KUKA KRL program: A_40mm_helical_45_10-LIN.src

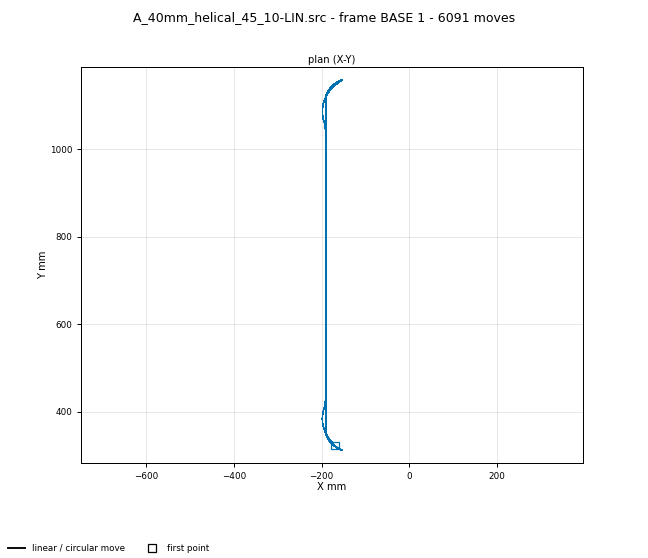
[picture p0: tool path of A_40mm_helical_45_10-LIN.src in frame BASE 1, 6091 of 6092 moves have a stored position in this frame; points joined in program order, loops and branches not executed]
&ACCESS RVP
DEF hoop( )

INTERRUPT DECL 3 WHEN $STOPMESS==TRUE DO IR_STOPM ( )
INTERRUPT ON 3
BAS (#INITMOV,0 )

ACTION(#AXIS_RESET,34,1000,#NOERROR,ERROR_CODE)
$H_POS=XHOME
PDAT_ACT=PDEFAULT
BAS (#PTP_DAT )
FDAT_ACT=FHOME
BAS (#FRAMES )
BAS (#VEL_PTP,100 )
PTP  XHOME
BAS(#TOOL,1)
BAS(#BASE,1)
LIN {X -170.340,Y +322.684,Z +0.000,A +20.000,E1 -17.457,E3 +0.000,E4 +0.000}
HALT
ACTION(#HUMM3_START,100,1000,#STOPONERROR,ERROR_CODE)
$APO.CDIS=85
$VEL_EXTAX[1]=100
LIN {X -175.568,Y +329.106,Z +0.000,A +20.000,E1 -24.747,E3 +17.234,E4 +0.000} C_DIS
LIN {X -184.074,Y +340.065,Z +0.000,A +20.000,E1 -33.664,E3 +40.174,E4 +0.000} C_DIS
LIN {X -190.779,Y +351.388,Z +0.000,A +20.000,E1 -40.083,E3 +57.952,E4 +0.000} C_DIS
LIN {X -195.254,Y +362.955,Z +0.000,A +20.000,E1 -44.515,E3 +72.705,E4 +0.000} C_DIS
LIN {X -197.754,Y +374.780,Z +0.000,A +20.000,E1 -47.450,E3 +86.127,E4 +0.000} C_DIS
LIN {X -198.310,Y +383.215,Z +0.000,A +19.956,E1 -48.698,E3 +95.251,E4 +0.000} C_DIS
LIN {X -197.912,Y +391.275,Z +0.000,A +18.601,E1 -49.158,E3 +103.969,E4 +0.000} C_DIS
LIN {X -196.679,Y +398.944,Z +0.000,A +13.989,E1 -48.784,E3 +112.523,E4 +0.000} C_DIS
LIN {X -194.742,Y +406.288,Z +0.000,A +8.476,E1 -48.001,E3 +121.206,E4 +0.000} C_DIS
LIN {X -192.748,Y +413.472,Z +0.000,A +3.905,E1 -47.267,E3 +130.216,E4 +0.000} C_DIS
LIN {X -191.781,Y +419.162,Z +0.000,A +1.739,E1 -46.975,E3 +137.484,E4 +0.000} C_DIS
LIN {X -190.795,Y +430.646,Z +0.000,A +0.152,E1 -46.707,E3 +152.145,E4 +0.000} C_DIS
LIN {X -190.395,Y +441.145,Z +0.000,A +0.001,E1 -46.583,E3 +165.538,E4 +0.000} C_DIS
LIN {X -190.239,Y +451.150,Z +0.000,A -0.000,E1 -46.528,E3 +178.306,E4 +0.000} C_DIS
LIN {X -190.161,Y +465.026,Z +0.000,A -0.000,E1 -46.506,E3 +196.021,E4 +0.000} C_DIS
LIN {X -190.142,Y +1057.148,Z +0.000,A -0.000,E1 -46.500,E3 +952.227,E4 +0.000} C_DIS
LIN {X -190.147,Y +1068.924,Z +0.000,A -0.000,E1 -46.499,E3 +967.268,E4 +0.000} C_DIS
LIN {X -190.159,Y +1079.072,Z +0.000,A -0.000,E1 -46.493,E3 +980.233,E4 +0.000} C_DIS
LIN {X -190.174,Y +1086.028,Z +0.000,A -0.000,E1 -46.483,E3 +989.127,E4 +0.000} C_DIS
LIN {X -190.200,Y +1096.186,Z +0.000,A -0.000,E1 -46.448,E3 +1002.131,E4 +0.000} C_DIS
LIN {X -190.154,Y +1108.998,Z +0.000,A -0.054,E1 -46.295,E3 +1018.626,E4 +0.000} C_DIS
LIN {X -189.772,Y +1119.341,Z +0.000,A -0.752,E1 -45.902,E3 +1032.164,E4 +0.000} C_DIS
LIN {X -189.097,Y +1124.276,Z +0.000,A -2.508,E1 -45.397,E3 +1038.896,E4 +0.000} C_DIS
LIN {X -187.410,Y +1129.069,Z +0.000,A -5.304,E1 -44.585,E3 +1046.069,E4 +0.000} C_DIS
LIN {X -183.899,Y +1134.873,Z +0.000,A -10.372,E1 -42.805,E3 +1056.075,E4 +0.000} C_DIS
LIN {X -179.711,Y +1140.065,Z +0.000,A -15.940,E1 -40.393,E3 +1066.861,E4 +0.000} C_DIS
LIN {X -176.763,Y +1143.197,Z +0.000,A -18.748,E1 -38.674,E3 +1074.599,E4 +0.000} C_DIS
LIN {X -172.185,Y +1147.423,Z +0.000,A -19.971,E1 -36.175,E3 +1087.329,E4 +0.000} C_DIS
LIN {X -165.999,Y +1152.127,Z +0.000,A -20.000,E1 -32.027,E3 +1107.087,E4 +0.000} C_DIS
LIN {X -160.138,Y +1155.667,Z +0.000,A -20.000,E1 -26.368,E3 +1131.457,E4 +0.000} C_DIS
LIN {X -155.625,Y +1157.756,Z +0.000,A -20.000,E1 -19.505,E3 +1160.133,E4 +0.000} C_DIS
LIN {X -153.552,Y +1158.113,Z +0.000,A -20.000,E1 -11.113,E3 +1195.884,E4 +0.000} C_DIS
LIN {X -156.311,Y +1155.540,Z +0.000,A -20.000,E1 -0.839,E3 +1239.244,E4 +0.000} C_DIS
LIN {X -161.281,Y +1151.851,Z +0.000,A -20.000,E1 +7.737,E3 +1269.143,E4 +0.000} C_DIS
LIN {X -167.493,Y +1147.157,Z +0.000,A -20.000,E1 +16.195,E3 +1293.582,E4 +0.000} C_DIS
LIN {X -173.235,Y +1142.221,Z +0.000,A -20.000,E1 +22.930,E3 +1310.884,E4 +0.000} C_DIS
LIN {X -181.123,Y +1133.734,Z +0.000,A -20.000,E1 +30.868,E3 +1331.640,E4 +0.000} C_DIS
LIN {X -189.654,Y +1120.856,Z +0.000,A -20.000,E1 +39.018,E3 +1353.654,E4 +0.000} C_DIS
LIN {X -195.246,Y +1107.046,Z +0.000,A -20.000,E1 +44.515,E3 +1371.556,E4 +0.000} C_DIS
LIN {X -198.051,Y +1092.368,Z +0.000,A -20.000,E1 +47.947,E3 +1388.082,E4 +0.000} C_DIS
LIN {X -198.143,Y +1081.370,Z +0.000,A -19.806,E1 +49.153,E3 +1399.943,E4 +0.000} C_DIS
LIN {X -197.177,Y +1073.569,Z +0.000,A -17.356,E1 +49.162,E3 +1408.527,E4 +0.000} C_DIS
LIN {X -195.448,Y +1066.139,Z +0.000,A -12.154,E1 +48.512,E3 +1417.122,E4 +0.000} C_DIS
LIN {X -193.346,Y +1058.941,Z +0.000,A -7.133,E1 +47.724,E3 +1426.002,E4 +0.000} C_DIS
LIN {X -191.781,Y +1050.839,Z +0.000,A -3.715,E1 +47.274,E3 +1436.335,E4 +0.000} C_DIS
LIN {X -190.795,Y +1039.355,Z +0.000,A -0.983,E1 +46.842,E3 +1450.995,E4 +0.000} C_DIS
LIN {X -190.395,Y +1028.856,Z +0.000,A -0.089,E1 +46.598,E3 +1464.389,E4 +0.000} C_DIS
LIN {X -190.239,Y +1018.851,Z +0.000,A -0.004,E1 +46.529,E3 +1477.157,E4 +0.000} C_DIS
LIN {X -190.161,Y +1004.975,Z +0.000,A +0.000,E1 +46.506,E3 +1494.871,E4 +0.000} C_DIS
LIN {X -190.142,Y +412.853,Z +0.000,A +0.000,E1 +46.501,E3 +2251.077,E4 +0.000} C_DIS
LIN {X -190.147,Y +401.077,Z +0.000,A +0.000,E1 +46.499,E3 +2266.118,E4 +0.000} C_DIS
LIN {X -190.159,Y +390.929,Z +0.000,A +0.000,E1 +46.494,E3 +2279.084,E4 +0.000} C_DIS
LIN {X -190.174,Y +383.973,Z +0.000,A +0.000,E1 +46.484,E3 +2287.977,E4 +0.000} C_DIS
LIN {X -190.200,Y +373.815,Z +0.000,A +0.000,E1 +46.448,E3 +2300.982,E4 +0.000} C_DIS
LIN {X -190.154,Y +361.003,Z +0.000,A +0.000,E1 +46.303,E3 +2317.476,E4 +0.000} C_DIS
LIN {X -189.772,Y +350.660,Z +0.000,A +0.049,E1 +45.996,E3 +2331.015,E4 +0.000} C_DIS
LIN {X -189.325,Y +346.917,Z +0.000,A +0.243,E1 +45.771,E3 +2336.084,E4 +0.000} C_DIS
LIN {X -188.196,Y +342.754,Z +0.000,A +1.966,E1 +45.249,E3 +2342.092,E4 +0.000} C_DIS
LIN {X -185.199,Y +337.023,Z +0.000,A +6.630,E1 +43.793,E3 +2351.466,E4 +0.000} C_DIS
LIN {X -181.141,Y +331.596,Z +0.000,A +12.274,E1 +41.569,E3 +2362.026,E4 +0.000} C_DIS
LIN {X -176.762,Y +326.804,Z +0.000,A +17.560,E1 +38.898,E3 +2373.450,E4 +0.000} C_DIS
LIN {X -172.184,Y +322.578,Z +0.000,A +19.859,E1 +36.197,E3 +2386.180,E4 +0.000} C_DIS
LIN {X -165.998,Y +317.874,Z +0.000,A +20.000,E1 +32.027,E3 +2405.938,E4 +0.000} C_DIS
LIN {X -160.137,Y +314.334,Z +0.000,A +20.000,E1 +26.368,E3 +2430.307,E4 +0.000} C_DIS
LIN {X -155.624,Y +312.245,Z +0.000,A +20.000,E1 +19.506,E3 +2458.983,E4 +0.000} C_DIS
LIN {X -153.557,Y +311.879,Z +0.000,A +20.000,E1 +11.113,E3 +2494.738,E4 +0.000} C_DIS
LIN {X -155.320,Y +313.348,Z +0.000,A +20.000,E1 +3.401,E3 +2527.922,E4 +0.000} C_DIS
LIN {X -160.005,Y +315.804,Z +0.000,A +20.000,E1 -4.720,E3 +2558.300,E4 +0.000} C_DIS
LIN {X -164.504,Y +318.255,Z +0.000,A +20.000,E1 -10.663,E3 +2577.669,E4 +0.000} C_DIS
LIN {X -170.340,Y +322.684,Z +0.000,A +20.000,E1 -17.457,E3 +2597.701,E4 +0.000} C_DIS
LIN {X -175.568,Y +329.106,Z +0.000,A +20.000,E1 -24.747,E3 +2614.935,E4 +0.000} C_DIS
LIN {X -184.074,Y +340.065,Z +0.000,A +20.000,E1 -33.664,E3 +2637.875,E4 +0.000} C_DIS
LIN {X -190.779,Y +351.388,Z +0.000,A +20.000,E1 -40.083,E3 +2655.653,E4 +0.000} C_DIS
LIN {X -195.254,Y +362.955,Z +0.000,A +20.000,E1 -44.515,E3 +2670.406,E4 +0.000} C_DIS
LIN {X -197.754,Y +374.780,Z +0.000,A +20.000,E1 -47.450,E3 +2683.828,E4 +0.000} C_DIS
LIN {X -198.310,Y +383.215,Z +0.000,A +19.956,E1 -48.698,E3 +2692.952,E4 +0.000} C_DIS
LIN {X -197.912,Y +391.275,Z +0.000,A +18.601,E1 -49.158,E3 +2701.670,E4 +0.000} C_DIS
LIN {X -196.679,Y +398.944,Z +0.000,A +13.989,E1 -48.784,E3 +2710.224,E4 +0.000} C_DIS
LIN {X -194.742,Y +406.288,Z +0.000,A +8.476,E1 -48.001,E3 +2718.907,E4 +0.000} C_DIS
LIN {X -192.748,Y +413.472,Z +0.000,A +3.905,E1 -47.267,E3 +2727.917,E4 +0.000} C_DIS
LIN {X -191.781,Y +419.162,Z +0.000,A +1.739,E1 -46.975,E3 +2735.185,E4 +0.000} C_DIS
LIN {X -190.795,Y +430.646,Z +0.000,A +0.152,E1 -46.707,E3 +2749.846,E4 +0.000} C_DIS
LIN {X -190.395,Y +441.145,Z +0.000,A +0.001,E1 -46.583,E3 +2763.239,E4 +0.000} C_DIS
LIN {X -190.239,Y +451.150,Z +0.000,A -0.000,E1 -46.528,E3 +2776.007,E4 +0.000} C_DIS
LIN {X -190.161,Y +465.026,Z +0.000,A -0.000,E1 -46.506,E3 +2793.722,E4 +0.000} C_DIS
LIN {X -190.142,Y +1057.148,Z +0.000,A -0.000,E1 -46.500,E3 +3549.928,E4 +0.000} C_DIS
LIN {X -190.147,Y +1068.924,Z +0.000,A -0.000,E1 -46.499,E3 +3564.969,E4 +0.000} C_DIS
LIN {X -190.159,Y +1079.072,Z +0.000,A -0.000,E1 -46.493,E3 +3577.934,E4 +0.000} C_DIS
LIN {X -190.174,Y +1086.028,Z +0.000,A -0.000,E1 -46.483,E3 +3586.828,E4 +0.000} C_DIS
LIN {X -190.200,Y +1096.186,Z +0.000,A -0.000,E1 -46.448,E3 +3599.832,E4 +0.000} C_DIS
LIN {X -190.154,Y +1108.998,Z +0.000,A -0.054,E1 -46.295,E3 +3616.327,E4 +0.000} C_DIS
LIN {X -189.772,Y +1119.341,Z +0.000,A -0.752,E1 -45.902,E3 +3629.865,E4 +0.000} C_DIS
LIN {X -189.097,Y +1124.276,Z +0.000,A -2.508,E1 -45.397,E3 +3636.597,E4 +0.000} C_DIS
LIN {X -187.410,Y +1129.069,Z +0.000,A -5.304,E1 -44.585,E3 +3643.770,E4 +0.000} C_DIS
LIN {X -183.899,Y +1134.873,Z +0.000,A -10.372,E1 -42.805,E3 +3653.776,E4 +0.000} C_DIS
LIN {X -179.711,Y +1140.065,Z +0.000,A -15.940,E1 -40.393,E3 +3664.562,E4 +0.000} C_DIS
LIN {X -176.763,Y +1143.197,Z +0.000,A -18.748,E1 -38.674,E3 +3672.300,E4 +0.000} C_DIS
LIN {X -172.185,Y +1147.423,Z +0.000,A -19.971,E1 -36.175,E3 +3685.030,E4 +0.000} C_DIS
LIN {X -165.999,Y +1152.127,Z +0.000,A -20.000,E1 -32.027,E3 +3704.788,E4 +0.000} C_DIS
LIN {X -160.138,Y +1155.667,Z +0.000,A -20.000,E1 -26.368,E3 +3729.158,E4 +0.000} C_DIS
LIN {X -155.625,Y +1157.756,Z +0.000,A -20.000,E1 -19.505,E3 +3757.834,E4 +0.000} C_DIS
LIN {X -153.552,Y +1158.113,Z +0.000,A -20.000,E1 -11.113,E3 +3793.585,E4 +0.000} C_DIS
LIN {X -156.311,Y +1155.540,Z +0.000,A -20.000,E1 -0.839,E3 +3836.945,E4 +0.000} C_DIS
LIN {X -161.281,Y +1151.851,Z +0.000,A -20.000,E1 +7.737,E3 +3866.844,E4 +0.000} C_DIS
LIN {X -167.493,Y +1147.157,Z +0.000,A -20.000,E1 +16.195,E3 +3891.283,E4 +0.000} C_DIS
LIN {X -173.235,Y +1142.221,Z +0.000,A -20.000,E1 +22.930,E3 +3908.585,E4 +0.000} C_DIS
LIN {X -181.123,Y +1133.734,Z +0.000,A -20.000,E1 +30.868,E3 +3929.341,E4 +0.000} C_DIS
LIN {X -189.654,Y +1120.856,Z +0.000,A -20.000,E1 +39.018,E3 +3951.355,E4 +0.000} C_DIS
LIN {X -195.246,Y +1107.046,Z +0.000,A -20.000,E1 +44.515,E3 +3969.257,E4 +0.000} C_DIS
LIN {X -198.051,Y +1092.368,Z +0.000,A -20.000,E1 +47.947,E3 +3985.783,E4 +0.000} C_DIS
LIN {X -198.143,Y +1081.370,Z +0.000,A -19.806,E1 +49.153,E3 +3997.644,E4 +0.000} C_DIS
LIN {X -197.177,Y +1073.569,Z +0.000,A -17.356,E1 +49.162,E3 +4006.228,E4 +0.000} C_DIS
LIN {X -195.448,Y +1066.139,Z +0.000,A -12.154,E1 +48.512,E3 +4014.823,E4 +0.000} C_DIS
LIN {X -193.346,Y +1058.941,Z +0.000,A -7.133,E1 +47.724,E3 +4023.703,E4 +0.000} C_DIS
LIN {X -191.781,Y +1050.839,Z +0.000,A -3.715,E1 +47.274,E3 +4034.036,E4 +0.000} C_DIS
LIN {X -190.795,Y +1039.355,Z +0.000,A -0.983,E1 +46.842,E3 +4048.696,E4 +0.000} C_DIS
LIN {X -190.395,Y +1028.856,Z +0.000,A -0.089,E1 +46.598,E3 +4062.090,E4 +0.000} C_DIS
LIN {X -190.239,Y +1018.851,Z +0.000,A -0.004,E1 +46.529,E3 +4074.858,E4 +0.000} C_DIS
LIN {X -190.161,Y +1004.975,Z +0.000,A +0.000,E1 +46.506,E3 +4092.572,E4 +0.000} C_DIS
LIN {X -190.142,Y +412.853,Z +0.000,A +0.000,E1 +46.501,E3 +4848.778,E4 +0.000} C_DIS
LIN {X -190.147,Y +401.077,Z +0.000,A +0.000,E1 +46.499,E3 +4863.819,E4 +0.000} C_DIS
LIN {X -190.159,Y +390.929,Z +0.000,A +0.000,E1 +46.494,E3 +4876.785,E4 +0.000} C_DIS
LIN {X -190.174,Y +383.973,Z +0.000,A +0.000,E1 +46.484,E3 +4885.678,E4 +0.000} C_DIS
LIN {X -190.200,Y +373.815,Z +0.000,A +0.000,E1 +46.448,E3 +4898.683,E4 +0.000} C_DIS
LIN {X -190.154,Y +361.003,Z +0.000,A +0.000,E1 +46.303,E3 +4915.177,E4 +0.000} C_DIS
LIN {X -189.772,Y +350.660,Z +0.000,A +0.049,E1 +45.996,E3 +4928.716,E4 +0.000} C_DIS
LIN {X -189.325,Y +346.917,Z +0.000,A +0.243,E1 +45.771,E3 +4933.785,E4 +0.000} C_DIS
LIN {X -188.196,Y +342.754,Z +0.000,A +1.966,E1 +45.249,E3 +4939.793,E4 +0.000} C_DIS
LIN {X -185.199,Y +337.023,Z +0.000,A +6.630,E1 +43.793,E3 +4949.167,E4 +0.000} C_DIS
LIN {X -181.141,Y +331.596,Z +0.000,A +12.274,E1 +41.569,E3 +4959.727,E4 +0.000} C_DIS
LIN {X -176.762,Y +326.804,Z +0.000,A +17.560,E1 +38.898,E3 +4971.151,E4 +0.000} C_DIS
LIN {X -172.184,Y +322.578,Z +0.000,A +19.859,E1 +36.197,E3 +4983.881,E4 +0.000} C_DIS
LIN {X -165.998,Y +317.874,Z +0.000,A +20.000,E1 +32.027,E3 +5003.639,E4 +0.000} C_DIS
LIN {X -160.137,Y +314.334,Z +0.000,A +20.000,E1 +26.368,E3 +5028.008,E4 +0.000} C_DIS
LIN {X -155.624,Y +312.245,Z +0.000,A +20.000,E1 +19.506,E3 +5056.684,E4 +0.000} C_DIS
LIN {X -153.557,Y +311.879,Z +0.000,A +20.000,E1 +11.113,E3 +5092.439,E4 +0.000} C_DIS
LIN {X -155.320,Y +313.348,Z +0.000,A +20.000,E1 +3.401,E3 +5125.623,E4 +0.000} C_DIS
LIN {X -160.005,Y +315.804,Z +0.000,A +20.000,E1 -4.720,E3 +5156.001,E4 +0.000} C_DIS
LIN {X -164.504,Y +318.255,Z +0.000,A +20.000,E1 -10.663,E3 +5175.370,E4 +0.000} C_DIS
LIN {X -170.340,Y +322.684,Z +0.000,A +20.000,E1 -17.457,E3 +5195.402,E4 +0.000} C_DIS
LIN {X -175.568,Y +329.106,Z +0.000,A +20.000,E1 -24.747,E3 +5212.636,E4 +0.000} C_DIS
LIN {X -184.074,Y +340.065,Z +0.000,A +20.000,E1 -33.664,E3 +5235.576,E4 +0.000} C_DIS
LIN {X -190.779,Y +351.388,Z +0.000,A +20.000,E1 -40.083,E3 +5253.354,E4 +0.000} C_DIS
LIN {X -195.254,Y +362.955,Z +0.000,A +20.000,E1 -44.515,E3 +5268.107,E4 +0.000} C_DIS
LIN {X -197.754,Y +374.780,Z +0.000,A +20.000,E1 -47.450,E3 +5281.529,E4 +0.000} C_DIS
LIN {X -198.310,Y +383.215,Z +0.000,A +19.956,E1 -48.698,E3 +5290.653,E4 +0.000} C_DIS
LIN {X -197.912,Y +391.275,Z +0.000,A +18.601,E1 -49.158,E3 +5299.371,E4 +0.000} C_DIS
LIN {X -196.679,Y +398.944,Z +0.000,A +13.989,E1 -48.784,E3 +5307.925,E4 +0.000} C_DIS
LIN {X -194.742,Y +406.288,Z +0.000,A +8.476,E1 -48.001,E3 +5316.608,E4 +0.000} C_DIS
LIN {X -192.748,Y +413.472,Z +0.000,A +3.905,E1 -47.267,E3 +5325.618,E4 +0.000} C_DIS
LIN {X -191.781,Y +419.162,Z +0.000,A +1.739,E1 -46.975,E3 +5332.886,E4 +0.000} C_DIS
LIN {X -190.795,Y +430.646,Z +0.000,A +0.152,E1 -46.707,E3 +5347.547,E4 +0.000} C_DIS
LIN {X -190.395,Y +441.145,Z +0.000,A +0.001,E1 -46.583,E3 +5360.940,E4 +0.000} C_DIS
LIN {X -190.239,Y +451.150,Z +0.000,A -0.000,E1 -46.528,E3 +5373.708,E4 +0.000} C_DIS
LIN {X -190.161,Y +465.026,Z +0.000,A -0.000,E1 -46.506,E3 +5391.423,E4 +0.000} C_DIS
LIN {X -190.142,Y +1057.148,Z +0.000,A -0.000,E1 -46.500,E3 +6147.629,E4 +0.000} C_DIS
LIN {X -190.147,Y +1068.924,Z +0.000,A -0.000,E1 -46.499,E3 +6162.670,E4 +0.000} C_DIS
LIN {X -190.159,Y +1079.072,Z +0.000,A -0.000,E1 -46.493,E3 +6175.635,E4 +0.000} C_DIS
LIN {X -190.174,Y +1086.028,Z +0.000,A -0.000,E1 -46.483,E3 +6184.529,E4 +0.000} C_DIS
LIN {X -190.200,Y +1096.186,Z +0.000,A -0.000,E1 -46.448,E3 +6197.533,E4 +0.000} C_DIS
LIN {X -190.154,Y +1108.998,Z +0.000,A -0.054,E1 -46.295,E3 +6214.028,E4 +0.000} C_DIS
LIN {X -189.772,Y +1119.341,Z +0.000,A -0.752,E1 -45.902,E3 +6227.566,E4 +0.000} C_DIS
LIN {X -189.097,Y +1124.276,Z +0.000,A -2.508,E1 -45.397,E3 +6234.298,E4 +0.000} C_DIS
LIN {X -187.410,Y +1129.069,Z +0.000,A -5.304,E1 -44.585,E3 +6241.471,E4 +0.000} C_DIS
LIN {X -183.899,Y +1134.873,Z +0.000,A -10.372,E1 -42.805,E3 +6251.477,E4 +0.000} C_DIS
LIN {X -179.711,Y +1140.065,Z +0.000,A -15.940,E1 -40.393,E3 +6262.263,E4 +0.000} C_DIS
LIN {X -176.763,Y +1143.197,Z +0.000,A -18.748,E1 -38.674,E3 +6270.001,E4 +0.000} C_DIS
LIN {X -172.185,Y +1147.423,Z +0.000,A -19.971,E1 -36.175,E3 +6282.731,E4 +0.000} C_DIS
LIN {X -165.999,Y +1152.127,Z +0.000,A -20.000,E1 -32.027,E3 +6302.489,E4 +0.000} C_DIS
LIN {X -160.138,Y +1155.667,Z +0.000,A -20.000,E1 -26.368,E3 +6326.859,E4 +0.000} C_DIS
LIN {X -155.625,Y +1157.756,Z +0.000,A -20.000,E1 -19.505,E3 +6355.535,E4 +0.000} C_DIS
LIN {X -153.552,Y +1158.113,Z +0.000,A -20.000,E1 -11.113,E3 +6391.286,E4 +0.000} C_DIS
LIN {X -156.311,Y +1155.540,Z +0.000,A -20.000,E1 -0.839,E3 +6434.646,E4 +0.000} C_DIS
LIN {X -161.281,Y +1151.851,Z +0.000,A -20.000,E1 +7.737,E3 +6464.545,E4 +0.000} C_DIS
LIN {X -167.493,Y +1147.157,Z +0.000,A -20.000,E1 +16.195,E3 +6488.984,E4 +0.000} C_DIS
LIN {X -173.235,Y +1142.221,Z +0.000,A -20.000,E1 +22.930,E3 +6506.286,E4 +0.000} C_DIS
LIN {X -181.123,Y +1133.734,Z +0.000,A -20.000,E1 +30.868,E3 +6527.042,E4 +0.000} C_DIS
LIN {X -189.654,Y +1120.856,Z +0.000,A -20.000,E1 +39.018,E3 +6549.056,E4 +0.000} C_DIS
LIN {X -195.246,Y +1107.046,Z +0.000,A -20.000,E1 +44.515,E3 +6566.958,E4 +0.000} C_DIS
LIN {X -198.051,Y +1092.368,Z +0.000,A -20.000,E1 +47.947,E3 +6583.484,E4 +0.000} C_DIS
LIN {X -198.143,Y +1081.370,Z +0.000,A -19.806,E1 +49.153,E3 +6595.345,E4 +0.000} C_DIS
LIN {X -197.177,Y +1073.569,Z +0.000,A -17.356,E1 +49.162,E3 +6603.929,E4 +0.000} C_DIS
LIN {X -195.448,Y +1066.139,Z +0.000,A -12.154,E1 +48.512,E3 +6612.524,E4 +0.000} C_DIS
LIN {X -193.346,Y +1058.941,Z +0.000,A -7.133,E1 +47.724,E3 +6621.404,E4 +0.000} C_DIS
LIN {X -191.781,Y +1050.839,Z +0.000,A -3.715,E1 +47.274,E3 +6631.737,E4 +0.000} C_DIS
LIN {X -190.795,Y +1039.355,Z +0.000,A -0.983,E1 +46.842,E3 +6646.397,E4 +0.000} C_DIS
LIN {X -190.395,Y +1028.856,Z +0.000,A -0.089,E1 +46.598,E3 +6659.791,E4 +0.000} C_DIS
LIN {X -190.239,Y +1018.851,Z +0.000,A -0.004,E1 +46.529,E3 +6672.559,E4 +0.000} C_DIS
LIN {X -190.161,Y +1004.975,Z +0.000,A +0.000,E1 +46.506,E3 +6690.273,E4 +0.000} C_DIS
LIN {X -190.142,Y +412.853,Z +0.000,A +0.000,E1 +46.501,E3 +7446.479,E4 +0.000} C_DIS
LIN {X -190.147,Y +401.077,Z +0.000,A +0.000,E1 +46.499,E3 +7461.520,E4 +0.000} C_DIS
LIN {X -190.159,Y +390.929,Z +0.000,A +0.000,E1 +46.494,E3 +7474.486,E4 +0.000} C_DIS
LIN {X -190.174,Y +383.973,Z +0.000,A +0.000,E1 +46.484,E3 +7483.379,E4 +0.000} C_DIS
LIN {X -190.200,Y +373.815,Z +0.000,A +0.000,E1 +46.448,E3 +7496.384,E4 +0.000} C_DIS
LIN {X -190.154,Y +361.003,Z +0.000,A +0.000,E1 +46.303,E3 +7512.878,E4 +0.000} C_DIS
LIN {X -189.772,Y +350.660,Z +0.000,A +0.049,E1 +45.996,E3 +7526.417,E4 +0.000} C_DIS
LIN {X -189.325,Y +346.917,Z +0.000,A +0.243,E1 +45.771,E3 +7531.486,E4 +0.000} C_DIS
LIN {X -188.196,Y +342.754,Z +0.000,A +1.966,E1 +45.249,E3 +7537.494,E4 +0.000} C_DIS
LIN {X -185.199,Y +337.023,Z +0.000,A +6.630,E1 +43.793,E3 +7546.868,E4 +0.000} C_DIS
LIN {X -181.141,Y +331.596,Z +0.000,A +12.274,E1 +41.569,E3 +7557.428,E4 +0.000} C_DIS
LIN {X -176.762,Y +326.804,Z +0.000,A +17.560,E1 +38.898,E3 +7568.852,E4 +0.000} C_DIS
LIN {X -172.184,Y +322.578,Z +0.000,A +19.859,E1 +36.197,E3 +7581.582,E4 +0.000} C_DIS
LIN {X -165.998,Y +317.874,Z +0.000,A +20.000,E1 +32.027,E3 +7601.340,E4 +0.000} C_DIS
LIN {X -160.137,Y +314.334,Z +0.000,A +20.000,E1 +26.368,E3 +7625.709,E4 +0.000} C_DIS
LIN {X -155.624,Y +312.245,Z +0.000,A +20.000,E1 +19.506,E3 +7654.385,E4 +0.000} C_DIS
LIN {X -153.557,Y +311.879,Z +0.000,A +20.000,E1 +11.113,E3 +7690.140,E4 +0.000} C_DIS
LIN {X -155.320,Y +313.348,Z +0.000,A +20.000,E1 +3.401,E3 +7723.324,E4 +0.000} C_DIS
LIN {X -160.005,Y +315.804,Z +0.000,A +20.000,E1 -4.720,E3 +7753.702,E4 +0.000} C_DIS
LIN {X -164.504,Y +318.255,Z +0.000,A +20.000,E1 -10.663,E3 +7773.071,E4 +0.000} C_DIS
LIN {X -170.340,Y +322.684,Z +0.000,A +20.000,E1 -17.457,E3 +7793.103,E4 +0.000} C_DIS
LIN {X -175.568,Y +329.106,Z +0.000,A +20.000,E1 -24.747,E3 +7810.337,E4 +0.000} C_DIS
LIN {X -184.074,Y +340.065,Z +0.000,A +20.000,E1 -33.664,E3 +7833.277,E4 +0.000} C_DIS
LIN {X -190.779,Y +351.388,Z +0.000,A +20.000,E1 -40.083,E3 +7851.055,E4 +0.000} C_DIS
LIN {X -195.254,Y +362.955,Z +0.000,A +20.000,E1 -44.515,E3 +7865.808,E4 +0.000} C_DIS
LIN {X -197.754,Y +374.780,Z +0.000,A +20.000,E1 -47.450,E3 +7879.230,E4 +0.000} C_DIS
LIN {X -198.310,Y +383.215,Z +0.000,A +19.956,E1 -48.698,E3 +7888.354,E4 +0.000} C_DIS
LIN {X -197.912,Y +391.275,Z +0.000,A +18.601,E1 -49.158,E3 +7897.072,E4 +0.000} C_DIS
LIN {X -196.679,Y +398.944,Z +0.000,A +13.989,E1 -48.784,E3 +7905.626,E4 +0.000} C_DIS
LIN {X -194.742,Y +406.288,Z +0.000,A +8.476,E1 -48.001,E3 +7914.309,E4 +0.000} C_DIS
LIN {X -192.748,Y +413.472,Z +0.000,A +3.905,E1 -47.267,E3 +7923.319,E4 +0.000} C_DIS
LIN {X -191.781,Y +419.162,Z +0.000,A +1.739,E1 -46.975,E3 +7930.587,E4 +0.000} C_DIS
LIN {X -190.795,Y +430.646,Z +0.000,A +0.152,E1 -46.707,E3 +7945.248,E4 +0.000} C_DIS
LIN {X -190.395,Y +441.145,Z +0.000,A +0.001,E1 -46.583,E3 +7958.641,E4 +0.000} C_DIS
LIN {X -190.239,Y +451.150,Z +0.000,A -0.000,E1 -46.528,E3 +7971.409,E4 +0.000} C_DIS
LIN {X -190.161,Y +465.026,Z +0.000,A -0.000,E1 -46.506,E3 +7989.124,E4 +0.000} C_DIS
LIN {X -190.142,Y +1057.148,Z +0.000,A -0.000,E1 -46.500,E3 +8745.330,E4 +0.000} C_DIS
LIN {X -190.147,Y +1068.924,Z +0.000,A -0.000,E1 -46.499,E3 +8760.371,E4 +0.000} C_DIS
LIN {X -190.159,Y +1079.072,Z +0.000,A -0.000,E1 -46.493,E3 +8773.336,E4 +0.000} C_DIS
LIN {X -190.174,Y +1086.028,Z +0.000,A -0.000,E1 -46.483,E3 +8782.230,E4 +0.000} C_DIS
LIN {X -190.200,Y +1096.186,Z +0.000,A -0.000,E1 -46.448,E3 +8795.234,E4 +0.000} C_DIS
LIN {X -190.154,Y +1108.998,Z +0.000,A -0.054,E1 -46.295,E3 +8811.729,E4 +0.000} C_DIS
LIN {X -189.772,Y +1119.341,Z +0.000,A -0.752,E1 -45.902,E3 +8825.267,E4 +0.000} C_DIS
LIN {X -189.097,Y +1124.276,Z +0.000,A -2.508,E1 -45.397,E3 +8831.999,E4 +0.000} C_DIS
LIN {X -187.410,Y +1129.069,Z +0.000,A -5.304,E1 -44.585,E3 +8839.172,E4 +0.000} C_DIS
LIN {X -183.899,Y +1134.873,Z +0.000,A -10.372,E1 -42.805,E3 +8849.178,E4 +0.000} C_DIS
LIN {X -179.711,Y +1140.065,Z +0.000,A -15.940,E1 -40.393,E3 +8859.964,E4 +0.000} C_DIS
LIN {X -176.763,Y +1143.197,Z +0.000,A -18.748,E1 -38.674,E3 +8867.702,E4 +0.000} C_DIS
LIN {X -172.185,Y +1147.423,Z +0.000,A -19.971,E1 -36.175,E3 +8880.432,E4 +0.000} C_DIS
LIN {X -165.999,Y +1152.127,Z +0.000,A -20.000,E1 -32.027,E3 +8900.190,E4 +0.000} C_DIS
LIN {X -160.138,Y +1155.667,Z +0.000,A -20.000,E1 -26.368,E3 +8924.560,E4 +0.000} C_DIS
LIN {X -155.625,Y +1157.756,Z +0.000,A -20.000,E1 -19.505,E3 +8953.236,E4 +0.000} C_DIS
LIN {X -153.552,Y +1158.113,Z +0.000,A -20.000,E1 -11.113,E3 +8988.987,E4 +0.000} C_DIS
LIN {X -156.311,Y +1155.540,Z +0.000,A -20.000,E1 -0.839,E3 +9032.347,E4 +0.000} C_DIS
LIN {X -161.281,Y +1151.851,Z +0.000,A -20.000,E1 +7.737,E3 +9062.246,E4 +0.000} C_DIS
LIN {X -167.493,Y +1147.157,Z +0.000,A -20.000,E1 +16.195,E3 +9086.685,E4 +0.000} C_DIS
LIN {X -173.235,Y +1142.221,Z +0.000,A -20.000,E1 +22.930,E3 +9103.987,E4 +0.000} C_DIS
LIN {X -181.123,Y +1133.734,Z +0.000,A -20.000,E1 +30.868,E3 +9124.743,E4 +0.000} C_DIS
LIN {X -189.654,Y +1120.856,Z +0.000,A -20.000,E1 +39.018,E3 +9146.757,E4 +0.000} C_DIS
LIN {X -195.246,Y +1107.046,Z +0.000,A -20.000,E1 +44.515,E3 +9164.659,E4 +0.000} C_DIS
LIN {X -198.051,Y +1092.368,Z +0.000,A -20.000,E1 +47.947,E3 +9181.185,E4 +0.000} C_DIS
LIN {X -198.143,Y +1081.370,Z +0.000,A -19.806,E1 +49.153,E3 +9193.046,E4 +0.000} C_DIS
LIN {X -197.177,Y +1073.569,Z +0.000,A -17.356,E1 +49.162,E3 +9201.630,E4 +0.000} C_DIS
LIN {X -195.448,Y +1066.139,Z +0.000,A -12.154,E1 +48.512,E3 +9210.225,E4 +0.000} C_DIS
LIN {X -193.346,Y +1058.941,Z +0.000,A -7.133,E1 +47.724,E3 +9219.105,E4 +0.000} C_DIS
LIN {X -191.781,Y +1050.839,Z +0.000,A -3.715,E1 +47.274,E3 +9229.438,E4 +0.000} C_DIS
LIN {X -190.795,Y +1039.355,Z +0.000,A -0.983,E1 +46.842,E3 +9244.098,E4 +0.000} C_DIS
LIN {X -190.395,Y +1028.856,Z +0.000,A -0.089,E1 +46.598,E3 +9257.492,E4 +0.000} C_DIS
LIN {X -190.239,Y +1018.851,Z +0.000,A -0.004,E1 +46.529,E3 +9270.260,E4 +0.000} C_DIS
LIN {X -190.161,Y +1004.975,Z +0.000,A +0.000,E1 +46.506,E3 +9287.974,E4 +0.000} C_DIS
LIN {X -190.142,Y +412.853,Z +0.000,A +0.000,E1 +46.501,E3 +10044.180,E4 +0.000} C_DIS
LIN {X -190.147,Y +401.077,Z +0.000,A +0.000,E1 +46.499,E3 +10059.221,E4 +0.000} C_DIS
LIN {X -190.159,Y +390.929,Z +0.000,A +0.000,E1 +46.494,E3 +10072.187,E4 +0.000} C_DIS
LIN {X -190.174,Y +383.973,Z +0.000,A +0.000,E1 +46.484,E3 +10081.080,E4 +0.000} C_DIS
LIN {X -190.200,Y +373.815,Z +0.000,A +0.000,E1 +46.448,E3 +10094.085,E4 +0.000} C_DIS
LIN {X -190.154,Y +361.003,Z +0.000,A +0.000,E1 +46.303,E3 +10110.579,E4 +0.000} C_DIS
LIN {X -189.772,Y +350.660,Z +0.000,A +0.049,E1 +45.996,E3 +10124.118,E4 +0.000} C_DIS
LIN {X -189.325,Y +346.917,Z +0.000,A +0.243,E1 +45.771,E3 +10129.187,E4 +0.000} C_DIS
LIN {X -188.196,Y +342.754,Z +0.000,A +1.966,E1 +45.249,E3 +10135.195,E4 +0.000} C_DIS
LIN {X -185.199,Y +337.023,Z +0.000,A +6.630,E1 +43.793,E3 +10144.569,E4 +0.000} C_DIS
LIN {X -181.141,Y +331.596,Z +0.000,A +12.274,E1 +41.569,E3 +10155.129,E4 +0.000} C_DIS
LIN {X -176.762,Y +326.804,Z +0.000,A +17.560,E1 +38.898,E3 +10166.553,E4 +0.000} C_DIS
LIN {X -172.184,Y +322.578,Z +0.000,A +19.859,E1 +36.197,E3 +10179.283,E4 +0.000} C_DIS
LIN {X -165.998,Y +317.874,Z +0.000,A +20.000,E1 +32.027,E3 +10199.041,E4 +0.000} C_DIS
LIN {X -160.137,Y +314.334,Z +0.000,A +20.000,E1 +26.368,E3 +10223.410,E4 +0.000} C_DIS
LIN {X -155.624,Y +312.245,Z +0.000,A +20.000,E1 +19.506,E3 +10252.086,E4 +0.000} C_DIS
LIN {X -153.557,Y +311.879,Z +0.000,A +20.000,E1 +11.113,E3 +10287.841,E4 +0.000} C_DIS
LIN {X -155.320,Y +313.348,Z +0.000,A +20.000,E1 +3.401,E3 +10321.025,E4 +0.000} C_DIS
LIN {X -160.005,Y +315.804,Z +0.000,A +20.000,E1 -4.720,E3 +10351.403,E4 +0.000} C_DIS
LIN {X -164.504,Y +318.255,Z +0.000,A +20.000,E1 -10.663,E3 +10370.772,E4 +0.000} C_DIS
LIN {X -170.340,Y +322.684,Z +0.000,A +20.000,E1 -17.457,E3 +10390.804,E4 +0.000} C_DIS
LIN {X -175.568,Y +329.106,Z +0.000,A +20.000,E1 -24.747,E3 +10408.038,E4 +0.000} C_DIS
LIN {X -184.074,Y +340.065,Z +0.000,A +20.000,E1 -33.664,E3 +10430.978,E4 +0.000} C_DIS
LIN {X -190.779,Y +351.388,Z +0.000,A +20.000,E1 -40.083,E3 +10448.756,E4 +0.000} C_DIS
LIN {X -195.254,Y +362.955,Z +0.000,A +20.000,E1 -44.515,E3 +10463.509,E4 +0.000} C_DIS
LIN {X -197.754,Y +374.780,Z +0.000,A +20.000,E1 -47.450,E3 +10476.931,E4 +0.000} C_DIS
LIN {X -198.310,Y +383.215,Z +0.000,A +19.956,E1 -48.698,E3 +10486.055,E4 +0.000} C_DIS
LIN {X -197.912,Y +391.275,Z +0.000,A +18.601,E1 -49.158,E3 +10494.773,E4 +0.000} C_DIS
LIN {X -196.679,Y +398.944,Z +0.000,A +13.989,E1 -48.784,E3 +10503.327,E4 +0.000} C_DIS
LIN {X -194.742,Y +406.288,Z +0.000,A +8.476,E1 -48.001,E3 +10512.010,E4 +0.000} C_DIS
LIN {X -192.748,Y +413.472,Z +0.000,A +3.905,E1 -47.267,E3 +10521.020,E4 +0.000} C_DIS
LIN {X -191.781,Y +419.162,Z +0.000,A +1.739,E1 -46.975,E3 +10528.288,E4 +0.000} C_DIS
LIN {X -190.795,Y +430.646,Z +0.000,A +0.152,E1 -46.707,E3 +10542.949,E4 +0.000} C_DIS
LIN {X -190.395,Y +441.145,Z +0.000,A +0.001,E1 -46.583,E3 +10556.342,E4 +0.000} C_DIS
LIN {X -190.239,Y +451.150,Z +0.000,A -0.000,E1 -46.528,E3 +10569.110,E4 +0.000} C_DIS
LIN {X -190.161,Y +465.026,Z +0.000,A -0.000,E1 -46.506,E3 +10586.825,E4 +0.000} C_DIS
LIN {X -190.142,Y +1057.148,Z +0.000,A -0.000,E1 -46.500,E3 +11343.031,E4 +0.000} C_DIS
LIN {X -190.147,Y +1068.924,Z +0.000,A -0.000,E1 -46.499,E3 +11358.072,E4 +0.000} C_DIS
LIN {X -190.159,Y +1079.072,Z +0.000,A -0.000,E1 -46.493,E3 +11371.037,E4 +0.000} C_DIS
LIN {X -190.174,Y +1086.028,Z +0.000,A -0.000,E1 -46.483,E3 +11379.931,E4 +0.000} C_DIS
LIN {X -190.200,Y +1096.186,Z +0.000,A -0.000,E1 -46.448,E3 +11392.935,E4 +0.000} C_DIS
LIN {X -190.154,Y +1108.998,Z +0.000,A -0.054,E1 -46.295,E3 +11409.430,E4 +0.000} C_DIS
LIN {X -189.772,Y +1119.341,Z +0.000,A -0.752,E1 -45.902,E3 +11422.968,E4 +0.000} C_DIS
LIN {X -189.097,Y +1124.276,Z +0.000,A -2.508,E1 -45.397,E3 +11429.700,E4 +0.000} C_DIS
LIN {X -187.410,Y +1129.069,Z +0.000,A -5.304,E1 -44.585,E3 +11436.873,E4 +0.000} C_DIS
LIN {X -183.899,Y +1134.873,Z +0.000,A -10.372,E1 -42.805,E3 +11446.879,E4 +0.000} C_DIS
LIN {X -179.711,Y +1140.065,Z +0.000,A -15.940,E1 -40.393,E3 +11457.665,E4 +0.000} C_DIS
LIN {X -176.763,Y +1143.197,Z +0.000,A -18.748,E1 -38.674,E3 +11465.403,E4 +0.000} C_DIS
LIN {X -172.185,Y +1147.423,Z +0.000,A -19.971,E1 -36.175,E3 +11478.133,E4 +0.000} C_DIS
LIN {X -165.999,Y +1152.127,Z +0.000,A -20.000,E1 -32.027,E3 +11497.891,E4 +0.000} C_DIS
LIN {X -160.138,Y +1155.667,Z +0.000,A -20.000,E1 -26.368,E3 +11522.261,E4 +0.000} C_DIS
LIN {X -155.625,Y +1157.756,Z +0.000,A -20.000,E1 -19.505,E3 +11550.937,E4 +0.000} C_DIS
LIN {X -153.552,Y +1158.113,Z +0.000,A -20.000,E1 -11.113,E3 +11586.688,E4 +0.000} C_DIS
LIN {X -156.311,Y +1155.540,Z +0.000,A -20.000,E1 -0.839,E3 +11630.048,E4 +0.000} C_DIS
LIN {X -161.281,Y +1151.851,Z +0.000,A -20.000,E1 +7.737,E3 +11659.947,E4 +0.000} C_DIS
LIN {X -167.493,Y +1147.157,Z +0.000,A -20.000,E1 +16.195,E3 +11684.386,E4 +0.000} C_DIS
LIN {X -173.235,Y +1142.221,Z +0.000,A -20.000,E1 +22.930,E3 +11701.688,E4 +0.000} C_DIS
LIN {X -181.123,Y +1133.734,Z +0.000,A -20.000,E1 +30.868,E3 +11722.444,E4 +0.000} C_DIS
LIN {X -189.654,Y +1120.856,Z +0.000,A -20.000,E1 +39.018,E3 +11744.458,E4 +0.000} C_DIS
LIN {X -195.246,Y +1107.046,Z +0.000,A -20.000,E1 +44.515,E3 +11762.360,E4 +0.000} C_DIS
LIN {X -198.051,Y +1092.368,Z +0.000,A -20.000,E1 +47.947,E3 +11778.886,E4 +0.000} C_DIS
LIN {X -198.143,Y +1081.370,Z +0.000,A -19.806,E1 +49.153,E3 +11790.747,E4 +0.000} C_DIS
LIN {X -197.177,Y +1073.569,Z +0.000,A -17.356,E1 +49.162,E3 +11799.331,E4 +0.000} C_DIS
LIN {X -195.448,Y +1066.139,Z +0.000,A -12.154,E1 +48.512,E3 +11807.926,E4 +0.000} C_DIS
LIN {X -193.346,Y +1058.941,Z +0.000,A -7.133,E1 +47.724,E3 +11816.806,E4 +0.000} C_DIS
LIN {X -191.781,Y +1050.839,Z +0.000,A -3.715,E1 +47.274,E3 +11827.139,E4 +0.000} C_DIS
LIN {X -190.795,Y +1039.355,Z +0.000,A -0.983,E1 +46.842,E3 +11841.799,E4 +0.000} C_DIS
LIN {X -190.395,Y +1028.856,Z +0.000,A -0.089,E1 +46.598,E3 +11855.193,E4 +0.000} C_DIS
LIN {X -190.239,Y +1018.851,Z +0.000,A -0.004,E1 +46.529,E3 +11867.961,E4 +0.000} C_DIS
LIN {X -190.161,Y +1004.975,Z +0.000,A +0.000,E1 +46.506,E3 +11885.675,E4 +0.000} C_DIS
LIN {X -190.142,Y +412.853,Z +0.000,A +0.000,E1 +46.501,E3 +12641.881,E4 +0.000} C_DIS
LIN {X -190.147,Y +401.077,Z +0.000,A +0.000,E1 +46.499,E3 +12656.922,E4 +0.000} C_DIS
LIN {X -190.159,Y +390.929,Z +0.000,A +0.000,E1 +46.494,E3 +12669.888,E4 +0.000} C_DIS
LIN {X -190.174,Y +383.973,Z +0.000,A +0.000,E1 +46.484,E3 +12678.781,E4 +0.000} C_DIS
LIN {X -190.200,Y +373.815,Z +0.000,A +0.000,E1 +46.448,E3 +12691.786,E4 +0.000} C_DIS
LIN {X -190.154,Y +361.003,Z +0.000,A +0.000,E1 +46.303,E3 +12708.280,E4 +0.000} C_DIS
LIN {X -189.772,Y +350.660,Z +0.000,A +0.049,E1 +45.996,E3 +12721.819,E4 +0.000} C_DIS
LIN {X -189.325,Y +346.917,Z +0.000,A +0.243,E1 +45.771,E3 +12726.888,E4 +0.000} C_DIS
LIN {X -188.196,Y +342.754,Z +0.000,A +1.966,E1 +45.249,E3 +12732.896,E4 +0.000} C_DIS
LIN {X -185.199,Y +337.023,Z +0.000,A +6.630,E1 +43.793,E3 +12742.270,E4 +0.000} C_DIS
LIN {X -181.141,Y +331.596,Z +0.000,A +12.274,E1 +41.569,E3 +12752.830,E4 +0.000} C_DIS
LIN {X -176.762,Y +326.804,Z +0.000,A +17.560,E1 +38.898,E3 +12764.254,E4 +0.000} C_DIS
LIN {X -172.184,Y +322.578,Z +0.000,A +19.859,E1 +36.197,E3 +12776.984,E4 +0.000} C_DIS
LIN {X -165.998,Y +317.874,Z +0.000,A +20.000,E1 +32.027,E3 +12796.742,E4 +0.000} C_DIS
LIN {X -160.137,Y +314.334,Z +0.000,A +20.000,E1 +26.368,E3 +12821.111,E4 +0.000} C_DIS
LIN {X -155.624,Y +312.245,Z +0.000,A +20.000,E1 +19.506,E3 +12849.787,E4 +0.000} C_DIS
LIN {X -153.557,Y +311.879,Z +0.000,A +20.000,E1 +11.113,E3 +12885.542,E4 +0.000} C_DIS
LIN {X -155.320,Y +313.348,Z +0.000,A +20.000,E1 +3.401,E3 +12918.726,E4 +0.000} C_DIS
LIN {X -160.005,Y +315.804,Z +0.000,A +20.000,E1 -4.720,E3 +12949.104,E4 +0.000} C_DIS
LIN {X -164.504,Y +318.255,Z +0.000,A +20.000,E1 -10.663,E3 +12968.473,E4 +0.000} C_DIS
LIN {X -170.340,Y +322.684,Z +0.000,A +20.000,E1 -17.457,E3 +12988.505,E4 +0.000} C_DIS
LIN {X -175.568,Y +329.106,Z +0.000,A +20.000,E1 -24.747,E3 +13005.739,E4 +0.000} C_DIS
LIN {X -184.074,Y +340.065,Z +0.000,A +20.000,E1 -33.664,E3 +13028.679,E4 +0.000} C_DIS
LIN {X -190.779,Y +351.388,Z +0.000,A +20.000,E1 -40.083,E3 +13046.457,E4 +0.000} C_DIS
LIN {X -195.254,Y +362.955,Z +0.000,A +20.000,E1 -44.515,E3 +13061.210,E4 +0.000} C_DIS
LIN {X -197.754,Y +374.780,Z +0.000,A +20.000,E1 -47.450,E3 +13074.632,E4 +0.000} C_DIS
LIN {X -198.310,Y +383.215,Z +0.000,A +19.956,E1 -48.698,E3 +13083.756,E4 +0.000} C_DIS
LIN {X -197.912,Y +391.275,Z +0.000,A +18.601,E1 -49.158,E3 +13092.474,E4 +0.000} C_DIS
LIN {X -196.679,Y +398.944,Z +0.000,A +13.989,E1 -48.784,E3 +13101.028,E4 +0.000} C_DIS
LIN {X -194.742,Y +406.288,Z +0.000,A +8.476,E1 -48.001,E3 +13109.711,E4 +0.000} C_DIS
LIN {X -192.748,Y +413.472,Z +0.000,A +3.905,E1 -47.267,E3 +13118.721,E4 +0.000} C_DIS
LIN {X -191.781,Y +419.162,Z +0.000,A +1.739,E1 -46.975,E3 +13125.989,E4 +0.000} C_DIS
LIN {X -190.795,Y +430.646,Z +0.000,A +0.152,E1 -46.707,E3 +13140.650,E4 +0.000} C_DIS
LIN {X -190.395,Y +441.145,Z +0.000,A +0.001,E1 -46.583,E3 +13154.043,E4 +0.000} C_DIS
LIN {X -190.239,Y +451.150,Z +0.000,A -0.000,E1 -46.528,E3 +13166.811,E4 +0.000} C_DIS
LIN {X -190.161,Y +465.026,Z +0.000,A -0.000,E1 -46.506,E3 +13184.526,E4 +0.000} C_DIS
LIN {X -190.142,Y +1057.148,Z +0.000,A -0.000,E1 -46.500,E3 +13940.732,E4 +0.000} C_DIS
LIN {X -190.147,Y +1068.924,Z +0.000,A -0.000,E1 -46.499,E3 +13955.773,E4 +0.000} C_DIS
LIN {X -190.159,Y +1079.072,Z +0.000,A -0.000,E1 -46.493,E3 +13968.738,E4 +0.000} C_DIS
LIN {X -190.174,Y +1086.028,Z +0.000,A -0.000,E1 -46.483,E3 +13977.632,E4 +0.000} C_DIS
LIN {X -190.200,Y +1096.186,Z +0.000,A -0.000,E1 -46.448,E3 +13990.636,E4 +0.000} C_DIS
LIN {X -190.154,Y +1108.998,Z +0.000,A -0.054,E1 -46.295,E3 +14007.131,E4 +0.000} C_DIS
LIN {X -189.772,Y +1119.341,Z +0.000,A -0.752,E1 -45.902,E3 +14020.669,E4 +0.000} C_DIS
LIN {X -189.097,Y +1124.276,Z +0.000,A -2.508,E1 -45.397,E3 +14027.401,E4 +0.000} C_DIS
LIN {X -187.410,Y +1129.069,Z +0.000,A -5.304,E1 -44.585,E3 +14034.574,E4 +0.000} C_DIS
LIN {X -183.899,Y +1134.873,Z +0.000,A -10.372,E1 -42.805,E3 +14044.580,E4 +0.000} C_DIS
LIN {X -179.711,Y +1140.065,Z +0.000,A -15.940,E1 -40.393,E3 +14055.366,E4 +0.000} C_DIS
LIN {X -176.763,Y +1143.197,Z +0.000,A -18.748,E1 -38.674,E3 +14063.104,E4 +0.000} C_DIS
LIN {X -172.185,Y +1147.423,Z +0.000,A -19.971,E1 -36.175,E3 +14075.834,E4 +0.000} C_DIS
LIN {X -165.999,Y +1152.127,Z +0.000,A -20.000,E1 -32.027,E3 +14095.592,E4 +0.000} C_DIS
LIN {X -160.138,Y +1155.667,Z +0.000,A -20.000,E1 -26.368,E3 +14119.962,E4 +0.000} C_DIS
LIN {X -155.625,Y +1157.756,Z +0.000,A -20.000,E1 -19.505,E3 +14148.638,E4 +0.000} C_DIS
LIN {X -153.552,Y +1158.113,Z +0.000,A -20.000,E1 -11.113,E3 +14184.389,E4 +0.000} C_DIS
LIN {X -156.311,Y +1155.540,Z +0.000,A -20.000,E1 -0.839,E3 +14227.749,E4 +0.000} C_DIS
LIN {X -161.281,Y +1151.851,Z +0.000,A -20.000,E1 +7.737,E3 +14257.648,E4 +0.000} C_DIS
LIN {X -167.493,Y +1147.157,Z +0.000,A -20.000,E1 +16.195,E3 +14282.087,E4 +0.000} C_DIS
LIN {X -173.235,Y +1142.221,Z +0.000,A -20.000,E1 +22.930,E3 +14299.389,E4 +0.000} C_DIS
LIN {X -181.123,Y +1133.734,Z +0.000,A -20.000,E1 +30.868,E3 +14320.145,E4 +0.000} C_DIS
LIN {X -189.654,Y +1120.856,Z +0.000,A -20.000,E1 +39.018,E3 +14342.159,E4 +0.000} C_DIS
LIN {X -195.246,Y +1107.046,Z +0.000,A -20.000,E1 +44.515,E3 +14360.061,E4 +0.000} C_DIS
LIN {X -198.051,Y +1092.368,Z +0.000,A -20.000,E1 +47.947,E3 +14376.587,E4 +0.000} C_DIS
LIN {X -198.143,Y +1081.370,Z +0.000,A -19.806,E1 +49.153,E3 +14388.448,E4 +0.000} C_DIS
LIN {X -197.177,Y +1073.569,Z +0.000,A -17.356,E1 +49.162,E3 +14397.032,E4 +0.000} C_DIS
LIN {X -195.448,Y +1066.139,Z +0.000,A -12.154,E1 +48.512,E3 +14405.627,E4 +0.000} C_DIS
LIN {X -193.346,Y +1058.941,Z +0.000,A -7.133,E1 +47.724,E3 +14414.507,E4 +0.000} C_DIS
LIN {X -191.781,Y +1050.839,Z +0.000,A -3.715,E1 +47.274,E3 +14424.840,E4 +0.000} C_DIS
LIN {X -190.795,Y +1039.355,Z +0.000,A -0.983,E1 +46.842,E3 +14439.500,E4 +0.000} C_DIS
LIN {X -190.395,Y +1028.856,Z +0.000,A -0.089,E1 +46.598,E3 +14452.894,E4 +0.000} C_DIS
LIN {X -190.239,Y +1018.851,Z +0.000,A -0.004,E1 +46.529,E3 +14465.662,E4 +0.000} C_DIS
LIN {X -190.161,Y +1004.975,Z +0.000,A +0.000,E1 +46.506,E3 +14483.376,E4 +0.000} C_DIS
LIN {X -190.142,Y +412.853,Z +0.000,A +0.000,E1 +46.501,E3 +15239.582,E4 +0.000} C_DIS
LIN {X -190.147,Y +401.077,Z +0.000,A +0.000,E1 +46.499,E3 +15254.623,E4 +0.000} C_DIS
LIN {X -190.159,Y +390.929,Z +0.000,A +0.000,E1 +46.494,E3 +15267.589,E4 +0.000} C_DIS
LIN {X -190.174,Y +383.973,Z +0.000,A +0.000,E1 +46.484,E3 +15276.482,E4 +0.000} C_DIS
LIN {X -190.200,Y +373.815,Z +0.000,A +0.000,E1 +46.448,E3 +15289.487,E4 +0.000} C_DIS
LIN {X -190.154,Y +361.003,Z +0.000,A +0.000,E1 +46.303,E3 +15305.981,E4 +0.000} C_DIS
LIN {X -189.772,Y +350.660,Z +0.000,A +0.049,E1 +45.996,E3 +15319.520,E4 +0.000} C_DIS
LIN {X -189.325,Y +346.917,Z +0.000,A +0.243,E1 +45.771,E3 +15324.589,E4 +0.000} C_DIS
LIN {X -188.196,Y +342.754,Z +0.000,A +1.966,E1 +45.249,E3 +15330.597,E4 +0.000} C_DIS
LIN {X -185.199,Y +337.023,Z +0.000,A +6.630,E1 +43.793,E3 +15339.971,E4 +0.000} C_DIS
LIN {X -181.141,Y +331.596,Z +0.000,A +12.274,E1 +41.569,E3 +15350.531,E4 +0.000} C_DIS
LIN {X -176.762,Y +326.804,Z +0.000,A +17.560,E1 +38.898,E3 +15361.955,E4 +0.000} C_DIS
LIN {X -172.184,Y +322.578,Z +0.000,A +19.859,E1 +36.197,E3 +15374.685,E4 +0.000} C_DIS
LIN {X -165.998,Y +317.874,Z +0.000,A +20.000,E1 +32.027,E3 +15394.443,E4 +0.000} C_DIS
LIN {X -160.137,Y +314.334,Z +0.000,A +20.000,E1 +26.368,E3 +15418.812,E4 +0.000} C_DIS
LIN {X -155.624,Y +312.245,Z +0.000,A +20.000,E1 +19.506,E3 +15447.488,E4 +0.000} C_DIS
LIN {X -153.557,Y +311.879,Z +0.000,A +20.000,E1 +11.113,E3 +15483.243,E4 +0.000} C_DIS
LIN {X -155.320,Y +313.348,Z +0.000,A +20.000,E1 +3.401,E3 +15516.427,E4 +0.000} C_DIS
LIN {X -160.005,Y +315.804,Z +0.000,A +20.000,E1 -4.720,E3 +15546.805,E4 +0.000} C_DIS
LIN {X -164.504,Y +318.255,Z +0.000,A +20.000,E1 -10.663,E3 +15566.174,E4 +0.000} C_DIS
LIN {X -170.340,Y +322.684,Z +0.000,A +20.000,E1 -17.457,E3 +15586.206,E4 +0.000} C_DIS
LIN {X -175.568,Y +329.106,Z +0.000,A +20.000,E1 -24.747,E3 +15603.440,E4 +0.000} C_DIS
LIN {X -184.074,Y +340.065,Z +0.000,A +20.000,E1 -33.664,E3 +15626.380,E4 +0.000} C_DIS
LIN {X -190.779,Y +351.388,Z +0.000,A +20.000,E1 -40.083,E3 +15644.158,E4 +0.000} C_DIS
LIN {X -195.254,Y +362.955,Z +0.000,A +20.000,E1 -44.515,E3 +15658.911,E4 +0.000} C_DIS
LIN {X -197.754,Y +374.780,Z +0.000,A +20.000,E1 -47.450,E3 +15672.333,E4 +0.000} C_DIS
LIN {X -198.310,Y +383.215,Z +0.000,A +19.956,E1 -48.698,E3 +15681.457,E4 +0.000} C_DIS
LIN {X -197.912,Y +391.275,Z +0.000,A +18.601,E1 -49.158,E3 +15690.175,E4 +0.000} C_DIS
LIN {X -196.679,Y +398.944,Z +0.000,A +13.989,E1 -48.784,E3 +15698.729,E4 +0.000} C_DIS
LIN {X -194.742,Y +406.288,Z +0.000,A +8.476,E1 -48.001,E3 +15707.412,E4 +0.000} C_DIS
LIN {X -192.748,Y +413.472,Z +0.000,A +3.905,E1 -47.267,E3 +15716.422,E4 +0.000} C_DIS
LIN {X -191.781,Y +419.162,Z +0.000,A +1.739,E1 -46.975,E3 +15723.690,E4 +0.000} C_DIS
LIN {X -190.795,Y +430.646,Z +0.000,A +0.152,E1 -46.707,E3 +15738.351,E4 +0.000} C_DIS
LIN {X -190.395,Y +441.145,Z +0.000,A +0.001,E1 -46.583,E3 +15751.744,E4 +0.000} C_DIS
LIN {X -190.239,Y +451.150,Z +0.000,A -0.000,E1 -46.528,E3 +15764.512,E4 +0.000} C_DIS
LIN {X -190.161,Y +465.026,Z +0.000,A -0.000,E1 -46.506,E3 +15782.227,E4 +0.000} C_DIS
LIN {X -190.142,Y +1057.148,Z +0.000,A -0.000,E1 -46.500,E3 +16538.433,E4 +0.000} C_DIS
LIN {X -190.147,Y +1068.924,Z +0.000,A -0.000,E1 -46.499,E3 +16553.474,E4 +0.000} C_DIS
LIN {X -190.159,Y +1079.072,Z +0.000,A -0.000,E1 -46.493,E3 +16566.439,E4 +0.000} C_DIS
LIN {X -190.174,Y +1086.028,Z +0.000,A -0.000,E1 -46.483,E3 +16575.333,E4 +0.000} C_DIS
LIN {X -190.200,Y +1096.186,Z +0.000,A -0.000,E1 -46.448,E3 +16588.337,E4 +0.000} C_DIS
LIN {X -190.154,Y +1108.998,Z +0.000,A -0.054,E1 -46.295,E3 +16604.832,E4 +0.000} C_DIS
LIN {X -189.772,Y +1119.341,Z +0.000,A -0.752,E1 -45.902,E3 +16618.370,E4 +0.000} C_DIS
LIN {X -189.097,Y +1124.276,Z +0.000,A -2.508,E1 -45.397,E3 +16625.102,E4 +0.000} C_DIS
LIN {X -187.410,Y +1129.069,Z +0.000,A -5.304,E1 -44.585,E3 +16632.275,E4 +0.000} C_DIS
LIN {X -183.899,Y +1134.873,Z +0.000,A -10.372,E1 -42.805,E3 +16642.281,E4 +0.000} C_DIS
LIN {X -179.711,Y +1140.065,Z +0.000,A -15.940,E1 -40.393,E3 +16653.067,E4 +0.000} C_DIS
LIN {X -176.763,Y +1143.197,Z +0.000,A -18.748,E1 -38.674,E3 +16660.805,E4 +0.000} C_DIS
LIN {X -172.185,Y +1147.423,Z +0.000,A -19.971,E1 -36.175,E3 +16673.535,E4 +0.000} C_DIS
LIN {X -165.999,Y +1152.127,Z +0.000,A -20.000,E1 -32.027,E3 +16693.293,E4 +0.000} C_DIS
LIN {X -160.138,Y +1155.667,Z +0.000,A -20.000,E1 -26.368,E3 +16717.663,E4 +0.000} C_DIS
LIN {X -155.625,Y +1157.756,Z +0.000,A -20.000,E1 -19.505,E3 +16746.339,E4 +0.000} C_DIS
LIN {X -153.552,Y +1158.113,Z +0.000,A -20.000,E1 -11.113,E3 +16782.090,E4 +0.000} C_DIS
LIN {X -156.311,Y +1155.540,Z +0.000,A -20.000,E1 -0.839,E3 +16825.450,E4 +0.000} C_DIS
LIN {X -161.281,Y +1151.851,Z +0.000,A -20.000,E1 +7.737,E3 +16855.349,E4 +0.000} C_DIS
LIN {X -167.493,Y +1147.157,Z +0.000,A -20.000,E1 +16.195,E3 +16879.788,E4 +0.000} C_DIS
LIN {X -173.235,Y +1142.221,Z +0.000,A -20.000,E1 +22.930,E3 +16897.090,E4 +0.000} C_DIS
LIN {X -181.123,Y +1133.734,Z +0.000,A -20.000,E1 +30.868,E3 +16917.846,E4 +0.000} C_DIS
LIN {X -189.654,Y +1120.856,Z +0.000,A -20.000,E1 +39.018,E3 +16939.860,E4 +0.000} C_DIS
LIN {X -195.246,Y +1107.046,Z +0.000,A -20.000,E1 +44.515,E3 +16957.762,E4 +0.000} C_DIS
LIN {X -198.051,Y +1092.368,Z +0.000,A -20.000,E1 +47.947,E3 +16974.288,E4 +0.000} C_DIS
LIN {X -198.143,Y +1081.370,Z +0.000,A -19.806,E1 +49.153,E3 +16986.149,E4 +0.000} C_DIS
LIN {X -197.177,Y +1073.569,Z +0.000,A -17.356,E1 +49.162,E3 +16994.733,E4 +0.000} C_DIS
LIN {X -195.448,Y +1066.139,Z +0.000,A -12.154,E1 +48.512,E3 +17003.328,E4 +0.000} C_DIS
LIN {X -193.346,Y +1058.941,Z +0.000,A -7.133,E1 +47.724,E3 +17012.208,E4 +0.000} C_DIS
LIN {X -191.781,Y +1050.839,Z +0.000,A -3.715,E1 +47.274,E3 +17022.541,E4 +0.000} C_DIS
LIN {X -190.795,Y +1039.355,Z +0.000,A -0.983,E1 +46.842,E3 +17037.201,E4 +0.000} C_DIS
LIN {X -190.395,Y +1028.856,Z +0.000,A -0.089,E1 +46.598,E3 +17050.595,E4 +0.000} C_DIS
LIN {X -190.239,Y +1018.851,Z +0.000,A -0.004,E1 +46.529,E3 +17063.363,E4 +0.000} C_DIS
LIN {X -190.161,Y +1004.975,Z +0.000,A +0.000,E1 +46.506,E3 +17081.077,E4 +0.000} C_DIS
LIN {X -190.142,Y +412.853,Z +0.000,A +0.000,E1 +46.501,E3 +17837.283,E4 +0.000} C_DIS
LIN {X -190.147,Y +401.077,Z +0.000,A +0.000,E1 +46.499,E3 +17852.324,E4 +0.000} C_DIS
LIN {X -190.159,Y +390.929,Z +0.000,A +0.000,E1 +46.494,E3 +17865.290,E4 +0.000} C_DIS
LIN {X -190.174,Y +383.973,Z +0.000,A +0.000,E1 +46.484,E3 +17874.183,E4 +0.000} C_DIS
LIN {X -190.200,Y +373.815,Z +0.000,A +0.000,E1 +46.448,E3 +17887.188,E4 +0.000} C_DIS
LIN {X -190.154,Y +361.003,Z +0.000,A +0.000,E1 +46.303,E3 +17903.682,E4 +0.000} C_DIS
LIN {X -189.772,Y +350.660,Z +0.000,A +0.049,E1 +45.996,E3 +17917.221,E4 +0.000} C_DIS
LIN {X -189.325,Y +346.917,Z +0.000,A +0.243,E1 +45.771,E3 +17922.290,E4 +0.000} C_DIS
LIN {X -188.196,Y +342.754,Z +0.000,A +1.966,E1 +45.249,E3 +17928.298,E4 +0.000} C_DIS
LIN {X -185.199,Y +337.023,Z +0.000,A +6.630,E1 +43.793,E3 +17937.672,E4 +0.000} C_DIS
LIN {X -181.141,Y +331.596,Z +0.000,A +12.274,E1 +41.569,E3 +17948.232,E4 +0.000} C_DIS
LIN {X -176.762,Y +326.804,Z +0.000,A +17.560,E1 +38.898,E3 +17959.656,E4 +0.000} C_DIS
LIN {X -172.184,Y +322.578,Z +0.000,A +19.859,E1 +36.197,E3 +17972.386,E4 +0.000} C_DIS
LIN {X -165.998,Y +317.874,Z +0.000,A +20.000,E1 +32.027,E3 +17992.144,E4 +0.000} C_DIS
LIN {X -160.137,Y +314.334,Z +0.000,A +20.000,E1 +26.368,E3 +18016.513,E4 +0.000} C_DIS
LIN {X -155.624,Y +312.245,Z +0.000,A +20.000,E1 +19.506,E3 +18045.189,E4 +0.000} C_DIS
LIN {X -153.557,Y +311.879,Z +0.000,A +20.000,E1 +11.113,E3 +18080.944,E4 +0.000} C_DIS
LIN {X -155.320,Y +313.348,Z +0.000,A +20.000,E1 +3.401,E3 +18114.128,E4 +0.000} C_DIS
LIN {X -160.005,Y +315.804,Z +0.000,A +20.000,E1 -4.720,E3 +18144.506,E4 +0.000} C_DIS
LIN {X -164.504,Y +318.255,Z +0.000,A +20.000,E1 -10.663,E3 +18163.875,E4 +0.000} C_DIS
LIN {X -170.340,Y +322.684,Z +0.000,A +20.000,E1 -17.457,E3 +18183.907,E4 +0.000} C_DIS
LIN {X -175.568,Y +329.106,Z +0.000,A +20.000,E1 -24.747,E3 +18201.141,E4 +0.000} C_DIS
LIN {X -184.074,Y +340.065,Z +0.000,A +20.000,E1 -33.664,E3 +18224.081,E4 +0.000} C_DIS
LIN {X -190.779,Y +351.388,Z +0.000,A +20.000,E1 -40.083,E3 +18241.859,E4 +0.000} C_DIS
LIN {X -195.254,Y +362.955,Z +0.000,A +20.000,E1 -44.515,E3 +18256.612,E4 +0.000} C_DIS
LIN {X -197.754,Y +374.780,Z +0.000,A +20.000,E1 -47.450,E3 +18270.034,E4 +0.000} C_DIS
LIN {X -198.310,Y +383.215,Z +0.000,A +19.956,E1 -48.698,E3 +18279.158,E4 +0.000} C_DIS
LIN {X -197.912,Y +391.275,Z +0.000,A +18.601,E1 -49.158,E3 +18287.876,E4 +0.000} C_DIS
LIN {X -196.679,Y +398.944,Z +0.000,A +13.989,E1 -48.784,E3 +18296.430,E4 +0.000} C_DIS
LIN {X -194.742,Y +406.288,Z +0.000,A +8.476,E1 -48.001,E3 +18305.113,E4 +0.000} C_DIS
LIN {X -192.748,Y +413.472,Z +0.000,A +3.905,E1 -47.267,E3 +18314.123,E4 +0.000} C_DIS
LIN {X -191.781,Y +419.162,Z +0.000,A +1.739,E1 -46.975,E3 +18321.391,E4 +0.000} C_DIS
LIN {X -190.795,Y +430.646,Z +0.000,A +0.152,E1 -46.707,E3 +18336.052,E4 +0.000} C_DIS
LIN {X -190.395,Y +441.145,Z +0.000,A +0.001,E1 -46.583,E3 +18349.445,E4 +0.000} C_DIS
LIN {X -190.239,Y +451.150,Z +0.000,A -0.000,E1 -46.528,E3 +18362.213,E4 +0.000} C_DIS
LIN {X -190.161,Y +465.026,Z +0.000,A -0.000,E1 -46.506,E3 +18379.928,E4 +0.000} C_DIS
LIN {X -190.142,Y +1057.148,Z +0.000,A -0.000,E1 -46.500,E3 +19136.134,E4 +0.000} C_DIS
LIN {X -190.147,Y +1068.924,Z +0.000,A -0.000,E1 -46.499,E3 +19151.175,E4 +0.000} C_DIS
LIN {X -190.159,Y +1079.072,Z +0.000,A -0.000,E1 -46.493,E3 +19164.140,E4 +0.000} C_DIS
LIN {X -190.174,Y +1086.028,Z +0.000,A -0.000,E1 -46.483,E3 +19173.034,E4 +0.000} C_DIS
LIN {X -190.200,Y +1096.186,Z +0.000,A -0.000,E1 -46.448,E3 +19186.038,E4 +0.000} C_DIS
LIN {X -190.154,Y +1108.998,Z +0.000,A -0.054,E1 -46.295,E3 +19202.533,E4 +0.000} C_DIS
LIN {X -189.772,Y +1119.341,Z +0.000,A -0.752,E1 -45.902,E3 +19216.071,E4 +0.000} C_DIS
LIN {X -189.097,Y +1124.276,Z +0.000,A -2.508,E1 -45.397,E3 +19222.803,E4 +0.000} C_DIS
LIN {X -187.410,Y +1129.069,Z +0.000,A -5.304,E1 -44.585,E3 +19229.976,E4 +0.000} C_DIS
LIN {X -183.899,Y +1134.873,Z +0.000,A -10.372,E1 -42.805,E3 +19239.982,E4 +0.000} C_DIS
LIN {X -179.711,Y +1140.065,Z +0.000,A -15.940,E1 -40.393,E3 +19250.768,E4 +0.000} C_DIS
LIN {X -176.763,Y +1143.197,Z +0.000,A -18.748,E1 -38.674,E3 +19258.506,E4 +0.000} C_DIS
LIN {X -172.185,Y +1147.423,Z +0.000,A -19.971,E1 -36.175,E3 +19271.236,E4 +0.000} C_DIS
LIN {X -165.999,Y +1152.127,Z +0.000,A -20.000,E1 -32.027,E3 +19290.994,E4 +0.000} C_DIS
LIN {X -160.138,Y +1155.667,Z +0.000,A -20.000,E1 -26.368,E3 +19315.364,E4 +0.000} C_DIS
LIN {X -155.625,Y +1157.756,Z +0.000,A -20.000,E1 -19.505,E3 +19344.040,E4 +0.000} C_DIS
LIN {X -153.552,Y +1158.113,Z +0.000,A -20.000,E1 -11.113,E3 +19379.791,E4 +0.000} C_DIS
LIN {X -156.311,Y +1155.540,Z +0.000,A -20.000,E1 -0.839,E3 +19423.151,E4 +0.000} C_DIS
LIN {X -161.281,Y +1151.851,Z +0.000,A -20.000,E1 +7.737,E3 +19453.050,E4 +0.000} C_DIS
LIN {X -167.493,Y +1147.157,Z +0.000,A -20.000,E1 +16.195,E3 +19477.489,E4 +0.000} C_DIS
LIN {X -173.235,Y +1142.221,Z +0.000,A -20.000,E1 +22.930,E3 +19494.791,E4 +0.000} C_DIS
LIN {X -181.123,Y +1133.734,Z +0.000,A -20.000,E1 +30.868,E3 +19515.547,E4 +0.000} C_DIS
LIN {X -189.654,Y +1120.856,Z +0.000,A -20.000,E1 +39.018,E3 +19537.561,E4 +0.000} C_DIS
LIN {X -195.246,Y +1107.046,Z +0.000,A -20.000,E1 +44.515,E3 +19555.463,E4 +0.000} C_DIS
LIN {X -198.051,Y +1092.368,Z +0.000,A -20.000,E1 +47.947,E3 +19571.989,E4 +0.000} C_DIS
LIN {X -198.143,Y +1081.370,Z +0.000,A -19.806,E1 +49.153,E3 +19583.850,E4 +0.000} C_DIS
LIN {X -197.177,Y +1073.569,Z +0.000,A -17.356,E1 +49.162,E3 +19592.434,E4 +0.000} C_DIS
LIN {X -195.448,Y +1066.139,Z +0.000,A -12.154,E1 +48.512,E3 +19601.029,E4 +0.000} C_DIS
LIN {X -193.346,Y +1058.941,Z +0.000,A -7.133,E1 +47.724,E3 +19609.909,E4 +0.000} C_DIS
LIN {X -191.781,Y +1050.839,Z +0.000,A -3.715,E1 +47.274,E3 +19620.242,E4 +0.000} C_DIS
LIN {X -190.795,Y +1039.355,Z +0.000,A -0.983,E1 +46.842,E3 +19634.902,E4 +0.000} C_DIS
LIN {X -190.395,Y +1028.856,Z +0.000,A -0.089,E1 +46.598,E3 +19648.296,E4 +0.000} C_DIS
LIN {X -190.239,Y +1018.851,Z +0.000,A -0.004,E1 +46.529,E3 +19661.064,E4 +0.000} C_DIS
LIN {X -190.161,Y +1004.975,Z +0.000,A +0.000,E1 +46.506,E3 +19678.778,E4 +0.000} C_DIS
LIN {X -190.142,Y +412.853,Z +0.000,A +0.000,E1 +46.501,E3 +20434.984,E4 +0.000} C_DIS
LIN {X -190.147,Y +401.077,Z +0.000,A +0.000,E1 +46.499,E3 +20450.025,E4 +0.000} C_DIS
LIN {X -190.159,Y +390.929,Z +0.000,A +0.000,E1 +46.494,E3 +20462.991,E4 +0.000} C_DIS
LIN {X -190.174,Y +383.973,Z +0.000,A +0.000,E1 +46.484,E3 +20471.884,E4 +0.000} C_DIS
LIN {X -190.200,Y +373.815,Z +0.000,A +0.000,E1 +46.448,E3 +20484.889,E4 +0.000} C_DIS
LIN {X -190.154,Y +361.003,Z +0.000,A +0.000,E1 +46.303,E3 +20501.383,E4 +0.000} C_DIS
LIN {X -189.772,Y +350.660,Z +0.000,A +0.049,E1 +45.996,E3 +20514.922,E4 +0.000} C_DIS
LIN {X -189.325,Y +346.917,Z +0.000,A +0.243,E1 +45.771,E3 +20519.991,E4 +0.000} C_DIS
LIN {X -188.196,Y +342.754,Z +0.000,A +1.966,E1 +45.249,E3 +20525.999,E4 +0.000} C_DIS
LIN {X -185.199,Y +337.023,Z +0.000,A +6.630,E1 +43.793,E3 +20535.373,E4 +0.000} C_DIS
LIN {X -181.141,Y +331.596,Z +0.000,A +12.274,E1 +41.569,E3 +20545.933,E4 +0.000} C_DIS
LIN {X -176.762,Y +326.804,Z +0.000,A +17.560,E1 +38.898,E3 +20557.357,E4 +0.000} C_DIS
LIN {X -172.184,Y +322.578,Z +0.000,A +19.859,E1 +36.197,E3 +20570.087,E4 +0.000} C_DIS
LIN {X -165.998,Y +317.874,Z +0.000,A +20.000,E1 +32.027,E3 +20589.845,E4 +0.000} C_DIS
LIN {X -160.137,Y +314.334,Z +0.000,A +20.000,E1 +26.368,E3 +20614.214,E4 +0.000} C_DIS
LIN {X -155.624,Y +312.245,Z +0.000,A +20.000,E1 +19.506,E3 +20642.890,E4 +0.000} C_DIS
LIN {X -153.557,Y +311.879,Z +0.000,A +20.000,E1 +11.113,E3 +20678.645,E4 +0.000} C_DIS
LIN {X -155.320,Y +313.348,Z +0.000,A +20.000,E1 +3.401,E3 +20711.829,E4 +0.000} C_DIS
LIN {X -160.005,Y +315.804,Z +0.000,A +20.000,E1 -4.720,E3 +20742.207,E4 +0.000} C_DIS
LIN {X -164.504,Y +318.255,Z +0.000,A +20.000,E1 -10.663,E3 +20761.576,E4 +0.000} C_DIS
LIN {X -170.340,Y +322.684,Z +0.000,A +20.000,E1 -17.457,E3 +20781.608,E4 +0.000} C_DIS
LIN {X -175.568,Y +329.106,Z +0.000,A +20.000,E1 -24.747,E3 +20798.842,E4 +0.000} C_DIS
LIN {X -184.074,Y +340.065,Z +0.000,A +20.000,E1 -33.664,E3 +20821.782,E4 +0.000} C_DIS
LIN {X -190.779,Y +351.388,Z +0.000,A +20.000,E1 -40.083,E3 +20839.560,E4 +0.000} C_DIS
LIN {X -195.254,Y +362.955,Z +0.000,A +20.000,E1 -44.515,E3 +20854.313,E4 +0.000} C_DIS
LIN {X -197.754,Y +374.780,Z +0.000,A +20.000,E1 -47.450,E3 +20867.735,E4 +0.000} C_DIS
LIN {X -198.310,Y +383.215,Z +0.000,A +19.956,E1 -48.698,E3 +20876.859,E4 +0.000} C_DIS
LIN {X -197.912,Y +391.275,Z +0.000,A +18.601,E1 -49.158,E3 +20885.577,E4 +0.000} C_DIS
LIN {X -196.679,Y +398.944,Z +0.000,A +13.989,E1 -48.784,E3 +20894.131,E4 +0.000} C_DIS
LIN {X -194.742,Y +406.288,Z +0.000,A +8.476,E1 -48.001,E3 +20902.814,E4 +0.000} C_DIS
LIN {X -192.748,Y +413.472,Z +0.000,A +3.905,E1 -47.267,E3 +20911.824,E4 +0.000} C_DIS
LIN {X -191.781,Y +419.162,Z +0.000,A +1.739,E1 -46.975,E3 +20919.092,E4 +0.000} C_DIS
LIN {X -190.795,Y +430.646,Z +0.000,A +0.152,E1 -46.707,E3 +20933.753,E4 +0.000} C_DIS
LIN {X -190.395,Y +441.145,Z +0.000,A +0.001,E1 -46.583,E3 +20947.146,E4 +0.000} C_DIS
LIN {X -190.239,Y +451.150,Z +0.000,A -0.000,E1 -46.528,E3 +20959.914,E4 +0.000} C_DIS
LIN {X -190.161,Y +465.026,Z +0.000,A -0.000,E1 -46.506,E3 +20977.629,E4 +0.000} C_DIS
LIN {X -190.142,Y +1057.148,Z +0.000,A -0.000,E1 -46.500,E3 +21733.835,E4 +0.000} C_DIS
LIN {X -190.147,Y +1068.924,Z +0.000,A -0.000,E1 -46.499,E3 +21748.876,E4 +0.000} C_DIS
LIN {X -190.159,Y +1079.072,Z +0.000,A -0.000,E1 -46.493,E3 +21761.841,E4 +0.000} C_DIS
LIN {X -190.174,Y +1086.028,Z +0.000,A -0.000,E1 -46.483,E3 +21770.735,E4 +0.000} C_DIS
LIN {X -190.200,Y +1096.186,Z +0.000,A -0.000,E1 -46.448,E3 +21783.739,E4 +0.000} C_DIS
LIN {X -190.154,Y +1108.998,Z +0.000,A -0.054,E1 -46.295,E3 +21800.234,E4 +0.000} C_DIS
LIN {X -189.772,Y +1119.341,Z +0.000,A -0.752,E1 -45.902,E3 +21813.772,E4 +0.000} C_DIS
LIN {X -189.097,Y +1124.276,Z +0.000,A -2.508,E1 -45.397,E3 +21820.504,E4 +0.000} C_DIS
LIN {X -187.410,Y +1129.069,Z +0.000,A -5.304,E1 -44.585,E3 +21827.677,E4 +0.000} C_DIS
LIN {X -183.899,Y +1134.873,Z +0.000,A -10.372,E1 -42.805,E3 +21837.683,E4 +0.000} C_DIS
LIN {X -179.711,Y +1140.065,Z +0.000,A -15.940,E1 -40.393,E3 +21848.469,E4 +0.000} C_DIS
LIN {X -176.763,Y +1143.197,Z +0.000,A -18.748,E1 -38.674,E3 +21856.207,E4 +0.000} C_DIS
LIN {X -172.185,Y +1147.423,Z +0.000,A -19.971,E1 -36.175,E3 +21868.937,E4 +0.000} C_DIS
LIN {X -165.999,Y +1152.127,Z +0.000,A -20.000,E1 -32.027,E3 +21888.695,E4 +0.000} C_DIS
LIN {X -160.138,Y +1155.667,Z +0.000,A -20.000,E1 -26.368,E3 +21913.065,E4 +0.000} C_DIS
LIN {X -155.625,Y +1157.756,Z +0.000,A -20.000,E1 -19.505,E3 +21941.741,E4 +0.000} C_DIS
LIN {X -153.552,Y +1158.113,Z +0.000,A -20.000,E1 -11.113,E3 +21977.492,E4 +0.000} C_DIS
LIN {X -156.311,Y +1155.540,Z +0.000,A -20.000,E1 -0.839,E3 +22020.852,E4 +0.000} C_DIS
LIN {X -161.281,Y +1151.851,Z +0.000,A -20.000,E1 +7.737,E3 +22050.751,E4 +0.000} C_DIS
LIN {X -167.493,Y +1147.157,Z +0.000,A -20.000,E1 +16.195,E3 +22075.190,E4 +0.000} C_DIS
LIN {X -173.235,Y +1142.221,Z +0.000,A -20.000,E1 +22.930,E3 +22092.492,E4 +0.000} C_DIS
LIN {X -181.123,Y +1133.734,Z +0.000,A -20.000,E1 +30.868,E3 +22113.248,E4 +0.000} C_DIS
LIN {X -189.654,Y +1120.856,Z +0.000,A -20.000,E1 +39.018,E3 +22135.262,E4 +0.000} C_DIS
LIN {X -195.246,Y +1107.046,Z +0.000,A -20.000,E1 +44.515,E3 +22153.164,E4 +0.000} C_DIS
LIN {X -198.051,Y +1092.368,Z +0.000,A -20.000,E1 +47.947,E3 +22169.690,E4 +0.000} C_DIS
LIN {X -198.143,Y +1081.370,Z +0.000,A -19.806,E1 +49.153,E3 +22181.551,E4 +0.000} C_DIS
LIN {X -197.177,Y +1073.569,Z +0.000,A -17.356,E1 +49.162,E3 +22190.135,E4 +0.000} C_DIS
LIN {X -195.448,Y +1066.139,Z +0.000,A -12.154,E1 +48.512,E3 +22198.730,E4 +0.000} C_DIS
LIN {X -193.346,Y +1058.941,Z +0.000,A -7.133,E1 +47.724,E3 +22207.610,E4 +0.000} C_DIS
LIN {X -191.781,Y +1050.839,Z +0.000,A -3.715,E1 +47.274,E3 +22217.943,E4 +0.000} C_DIS
LIN {X -190.795,Y +1039.355,Z +0.000,A -0.983,E1 +46.842,E3 +22232.603,E4 +0.000} C_DIS
LIN {X -190.395,Y +1028.856,Z +0.000,A -0.089,E1 +46.598,E3 +22245.997,E4 +0.000} C_DIS
LIN {X -190.239,Y +1018.851,Z +0.000,A -0.004,E1 +46.529,E3 +22258.765,E4 +0.000} C_DIS
LIN {X -190.161,Y +1004.975,Z +0.000,A +0.000,E1 +46.506,E3 +22276.479,E4 +0.000} C_DIS
LIN {X -190.142,Y +412.853,Z +0.000,A +0.000,E1 +46.501,E3 +23032.685,E4 +0.000} C_DIS
LIN {X -190.147,Y +401.077,Z +0.000,A +0.000,E1 +46.499,E3 +23047.726,E4 +0.000} C_DIS
LIN {X -190.159,Y +390.929,Z +0.000,A +0.000,E1 +46.494,E3 +23060.692,E4 +0.000} C_DIS
LIN {X -190.174,Y +383.973,Z +0.000,A +0.000,E1 +46.484,E3 +23069.585,E4 +0.000} C_DIS
LIN {X -190.200,Y +373.815,Z +0.000,A +0.000,E1 +46.448,E3 +23082.590,E4 +0.000} C_DIS
LIN {X -190.154,Y +361.003,Z +0.000,A +0.000,E1 +46.303,E3 +23099.084,E4 +0.000} C_DIS
LIN {X -189.772,Y +350.660,Z +0.000,A +0.049,E1 +45.996,E3 +23112.623,E4 +0.000} C_DIS
LIN {X -189.325,Y +346.917,Z +0.000,A +0.243,E1 +45.771,E3 +23117.692,E4 +0.000} C_DIS
LIN {X -188.196,Y +342.754,Z +0.000,A +1.966,E1 +45.249,E3 +23123.700,E4 +0.000} C_DIS
LIN {X -185.199,Y +337.023,Z +0.000,A +6.630,E1 +43.793,E3 +23133.074,E4 +0.000} C_DIS
LIN {X -181.141,Y +331.596,Z +0.000,A +12.274,E1 +41.569,E3 +23143.634,E4 +0.000} C_DIS
LIN {X -176.762,Y +326.804,Z +0.000,A +17.560,E1 +38.898,E3 +23155.058,E4 +0.000} C_DIS
LIN {X -172.184,Y +322.578,Z +0.000,A +19.859,E1 +36.197,E3 +23167.788,E4 +0.000} C_DIS
LIN {X -165.998,Y +317.874,Z +0.000,A +20.000,E1 +32.027,E3 +23187.546,E4 +0.000} C_DIS
LIN {X -160.137,Y +314.334,Z +0.000,A +20.000,E1 +26.368,E3 +23211.915,E4 +0.000} C_DIS
LIN {X -155.624,Y +312.245,Z +0.000,A +20.000,E1 +19.506,E3 +23240.591,E4 +0.000} C_DIS
LIN {X -153.557,Y +311.879,Z +0.000,A +20.000,E1 +11.113,E3 +23276.346,E4 +0.000} C_DIS
LIN {X -155.320,Y +313.348,Z +0.000,A +20.000,E1 +3.401,E3 +23309.530,E4 +0.000} C_DIS
LIN {X -160.005,Y +315.804,Z +0.000,A +20.000,E1 -4.720,E3 +23339.908,E4 +0.000} C_DIS
LIN {X -164.504,Y +318.255,Z +0.000,A +20.000,E1 -10.663,E3 +23359.277,E4 +0.000} C_DIS
LIN {X -170.340,Y +322.684,Z +0.000,A +20.000,E1 -17.457,E3 +23379.309,E4 +0.000} C_DIS
LIN {X -175.568,Y +329.106,Z +0.000,A +20.000,E1 -24.747,E3 +23396.543,E4 +0.000} C_DIS
LIN {X -184.074,Y +340.065,Z +0.000,A +20.000,E1 -33.664,E3 +23419.483,E4 +0.000} C_DIS
LIN {X -190.779,Y +351.388,Z +0.000,A +20.000,E1 -40.083,E3 +23437.261,E4 +0.000} C_DIS
LIN {X -195.254,Y +362.955,Z +0.000,A +20.000,E1 -44.515,E3 +23452.014,E4 +0.000} C_DIS
LIN {X -197.754,Y +374.780,Z +0.000,A +20.000,E1 -47.450,E3 +23465.436,E4 +0.000} C_DIS
LIN {X -198.310,Y +383.215,Z +0.000,A +19.956,E1 -48.698,E3 +23474.560,E4 +0.000} C_DIS
LIN {X -197.912,Y +391.275,Z +0.000,A +18.601,E1 -49.158,E3 +23483.278,E4 +0.000} C_DIS
LIN {X -196.679,Y +398.944,Z +0.000,A +13.989,E1 -48.784,E3 +23491.832,E4 +0.000} C_DIS
LIN {X -194.742,Y +406.288,Z +0.000,A +8.476,E1 -48.001,E3 +23500.515,E4 +0.000} C_DIS
LIN {X -192.748,Y +413.472,Z +0.000,A +3.905,E1 -47.267,E3 +23509.525,E4 +0.000} C_DIS
LIN {X -191.781,Y +419.162,Z +0.000,A +1.739,E1 -46.975,E3 +23516.793,E4 +0.000} C_DIS
LIN {X -190.795,Y +430.646,Z +0.000,A +0.152,E1 -46.707,E3 +23531.454,E4 +0.000} C_DIS
LIN {X -190.395,Y +441.145,Z +0.000,A +0.001,E1 -46.583,E3 +23544.847,E4 +0.000} C_DIS
LIN {X -190.239,Y +451.150,Z +0.000,A -0.000,E1 -46.528,E3 +23557.615,E4 +0.000} C_DIS
LIN {X -190.161,Y +465.026,Z +0.000,A -0.000,E1 -46.506,E3 +23575.330,E4 +0.000} C_DIS
LIN {X -190.142,Y +1057.148,Z +0.000,A -0.000,E1 -46.500,E3 +24331.536,E4 +0.000} C_DIS
LIN {X -190.147,Y +1068.924,Z +0.000,A -0.000,E1 -46.499,E3 +24346.577,E4 +0.000} C_DIS
LIN {X -190.159,Y +1079.072,Z +0.000,A -0.000,E1 -46.493,E3 +24359.542,E4 +0.000} C_DIS
LIN {X -190.174,Y +1086.028,Z +0.000,A -0.000,E1 -46.483,E3 +24368.436,E4 +0.000} C_DIS
LIN {X -190.200,Y +1096.186,Z +0.000,A -0.000,E1 -46.448,E3 +24381.440,E4 +0.000} C_DIS
LIN {X -190.154,Y +1108.998,Z +0.000,A -0.054,E1 -46.295,E3 +24397.935,E4 +0.000} C_DIS
LIN {X -189.772,Y +1119.341,Z +0.000,A -0.752,E1 -45.902,E3 +24411.473,E4 +0.000} C_DIS
LIN {X -189.097,Y +1124.276,Z +0.000,A -2.508,E1 -45.397,E3 +24418.205,E4 +0.000} C_DIS
LIN {X -187.410,Y +1129.069,Z +0.000,A -5.304,E1 -44.585,E3 +24425.378,E4 +0.000} C_DIS
LIN {X -183.899,Y +1134.873,Z +0.000,A -10.372,E1 -42.805,E3 +24435.384,E4 +0.000} C_DIS
LIN {X -179.711,Y +1140.065,Z +0.000,A -15.940,E1 -40.393,E3 +24446.170,E4 +0.000} C_DIS
LIN {X -176.763,Y +1143.197,Z +0.000,A -18.748,E1 -38.674,E3 +24453.908,E4 +0.000} C_DIS
LIN {X -172.185,Y +1147.423,Z +0.000,A -19.971,E1 -36.175,E3 +24466.638,E4 +0.000} C_DIS
LIN {X -165.999,Y +1152.127,Z +0.000,A -20.000,E1 -32.027,E3 +24486.396,E4 +0.000} C_DIS
LIN {X -160.138,Y +1155.667,Z +0.000,A -20.000,E1 -26.368,E3 +24510.766,E4 +0.000} C_DIS
LIN {X -155.625,Y +1157.756,Z +0.000,A -20.000,E1 -19.505,E3 +24539.442,E4 +0.000} C_DIS
LIN {X -153.552,Y +1158.113,Z +0.000,A -20.000,E1 -11.113,E3 +24575.193,E4 +0.000} C_DIS
LIN {X -156.311,Y +1155.540,Z +0.000,A -20.000,E1 -0.839,E3 +24618.553,E4 +0.000} C_DIS
LIN {X -161.281,Y +1151.851,Z +0.000,A -20.000,E1 +7.737,E3 +24648.452,E4 +0.000} C_DIS
LIN {X -167.493,Y +1147.157,Z +0.000,A -20.000,E1 +16.195,E3 +24672.891,E4 +0.000} C_DIS
LIN {X -173.235,Y +1142.221,Z +0.000,A -20.000,E1 +22.930,E3 +24690.193,E4 +0.000} C_DIS
LIN {X -181.123,Y +1133.734,Z +0.000,A -20.000,E1 +30.868,E3 +24710.949,E4 +0.000} C_DIS
LIN {X -189.654,Y +1120.856,Z +0.000,A -20.000,E1 +39.018,E3 +24732.963,E4 +0.000} C_DIS
LIN {X -195.246,Y +1107.046,Z +0.000,A -20.000,E1 +44.515,E3 +24750.865,E4 +0.000} C_DIS
LIN {X -198.051,Y +1092.368,Z +0.000,A -20.000,E1 +47.947,E3 +24767.391,E4 +0.000} C_DIS
LIN {X -198.143,Y +1081.370,Z +0.000,A -19.806,E1 +49.153,E3 +24779.252,E4 +0.000} C_DIS
LIN {X -197.177,Y +1073.569,Z +0.000,A -17.356,E1 +49.162,E3 +24787.836,E4 +0.000} C_DIS
LIN {X -195.448,Y +1066.139,Z +0.000,A -12.154,E1 +48.512,E3 +24796.431,E4 +0.000} C_DIS
LIN {X -193.346,Y +1058.941,Z +0.000,A -7.133,E1 +47.724,E3 +24805.311,E4 +0.000} C_DIS
LIN {X -191.781,Y +1050.839,Z +0.000,A -3.715,E1 +47.274,E3 +24815.644,E4 +0.000} C_DIS
LIN {X -190.795,Y +1039.355,Z +0.000,A -0.983,E1 +46.842,E3 +24830.304,E4 +0.000} C_DIS
LIN {X -190.395,Y +1028.856,Z +0.000,A -0.089,E1 +46.598,E3 +24843.698,E4 +0.000} C_DIS
LIN {X -190.239,Y +1018.851,Z +0.000,A -0.004,E1 +46.529,E3 +24856.466,E4 +0.000} C_DIS
LIN {X -190.161,Y +1004.975,Z +0.000,A +0.000,E1 +46.506,E3 +24874.180,E4 +0.000} C_DIS
LIN {X -190.142,Y +412.853,Z +0.000,A +0.000,E1 +46.501,E3 +25630.386,E4 +0.000} C_DIS
LIN {X -190.147,Y +401.077,Z +0.000,A +0.000,E1 +46.499,E3 +25645.427,E4 +0.000} C_DIS
LIN {X -190.159,Y +390.929,Z +0.000,A +0.000,E1 +46.494,E3 +25658.393,E4 +0.000} C_DIS
LIN {X -190.174,Y +383.973,Z +0.000,A +0.000,E1 +46.484,E3 +25667.286,E4 +0.000} C_DIS
LIN {X -190.200,Y +373.815,Z +0.000,A +0.000,E1 +46.448,E3 +25680.291,E4 +0.000} C_DIS
LIN {X -190.154,Y +361.003,Z +0.000,A +0.000,E1 +46.303,E3 +25696.785,E4 +0.000} C_DIS
LIN {X -189.772,Y +350.660,Z +0.000,A +0.049,E1 +45.996,E3 +25710.324,E4 +0.000} C_DIS
LIN {X -189.325,Y +346.917,Z +0.000,A +0.243,E1 +45.771,E3 +25715.393,E4 +0.000} C_DIS
LIN {X -188.196,Y +342.754,Z +0.000,A +1.966,E1 +45.249,E3 +25721.401,E4 +0.000} C_DIS
LIN {X -185.199,Y +337.023,Z +0.000,A +6.630,E1 +43.793,E3 +25730.775,E4 +0.000} C_DIS
LIN {X -181.141,Y +331.596,Z +0.000,A +12.274,E1 +41.569,E3 +25741.335,E4 +0.000} C_DIS
LIN {X -176.762,Y +326.804,Z +0.000,A +17.560,E1 +38.898,E3 +25752.759,E4 +0.000} C_DIS
LIN {X -172.184,Y +322.578,Z +0.000,A +19.859,E1 +36.197,E3 +25765.489,E4 +0.000} C_DIS
LIN {X -165.998,Y +317.874,Z +0.000,A +20.000,E1 +32.027,E3 +25785.247,E4 +0.000} C_DIS
LIN {X -160.137,Y +314.334,Z +0.000,A +20.000,E1 +26.368,E3 +25809.616,E4 +0.000} C_DIS
LIN {X -155.624,Y +312.245,Z +0.000,A +20.000,E1 +19.506,E3 +25838.292,E4 +0.000} C_DIS
LIN {X -153.557,Y +311.879,Z +0.000,A +20.000,E1 +11.113,E3 +25874.047,E4 +0.000} C_DIS
LIN {X -155.320,Y +313.348,Z +0.000,A +20.000,E1 +3.401,E3 +25907.231,E4 +0.000} C_DIS
LIN {X -160.005,Y +315.804,Z +0.000,A +20.000,E1 -4.720,E3 +25937.609,E4 +0.000} C_DIS
LIN {X -164.504,Y +318.255,Z +0.000,A +20.000,E1 -10.663,E3 +25956.978,E4 +0.000} C_DIS
LIN {X -170.340,Y +322.684,Z +0.000,A +20.000,E1 -17.457,E3 +25977.010,E4 +0.000} C_DIS
LIN {X -175.568,Y +329.106,Z +0.000,A +20.000,E1 -24.747,E3 +25994.244,E4 +0.000} C_DIS
LIN {X -184.074,Y +340.065,Z +0.000,A +20.000,E1 -33.664,E3 +26017.184,E4 +0.000} C_DIS
LIN {X -190.779,Y +351.388,Z +0.000,A +20.000,E1 -40.083,E3 +26034.962,E4 +0.000} C_DIS
LIN {X -195.254,Y +362.955,Z +0.000,A +20.000,E1 -44.515,E3 +26049.715,E4 +0.000} C_DIS
LIN {X -197.754,Y +374.780,Z +0.000,A +20.000,E1 -47.450,E3 +26063.137,E4 +0.000} C_DIS
LIN {X -198.310,Y +383.215,Z +0.000,A +19.956,E1 -48.698,E3 +26072.261,E4 +0.000} C_DIS
LIN {X -197.912,Y +391.275,Z +0.000,A +18.601,E1 -49.158,E3 +26080.979,E4 +0.000} C_DIS
LIN {X -196.679,Y +398.944,Z +0.000,A +13.989,E1 -48.784,E3 +26089.533,E4 +0.000} C_DIS
LIN {X -194.742,Y +406.288,Z +0.000,A +8.476,E1 -48.001,E3 +26098.216,E4 +0.000} C_DIS
LIN {X -192.748,Y +413.472,Z +0.000,A +3.905,E1 -47.267,E3 +26107.226,E4 +0.000} C_DIS
LIN {X -191.781,Y +419.162,Z +0.000,A +1.739,E1 -46.975,E3 +26114.494,E4 +0.000} C_DIS
LIN {X -190.795,Y +430.646,Z +0.000,A +0.152,E1 -46.707,E3 +26129.155,E4 +0.000} C_DIS
LIN {X -190.395,Y +441.145,Z +0.000,A +0.001,E1 -46.583,E3 +26142.548,E4 +0.000} C_DIS
LIN {X -190.239,Y +451.150,Z +0.000,A -0.000,E1 -46.528,E3 +26155.316,E4 +0.000} C_DIS
LIN {X -190.161,Y +465.026,Z +0.000,A -0.000,E1 -46.506,E3 +26173.031,E4 +0.000} C_DIS
LIN {X -190.142,Y +1057.148,Z +0.000,A -0.000,E1 -46.500,E3 +26929.237,E4 +0.000} C_DIS
LIN {X -190.147,Y +1068.924,Z +0.000,A -0.000,E1 -46.499,E3 +26944.278,E4 +0.000} C_DIS
LIN {X -190.159,Y +1079.072,Z +0.000,A -0.000,E1 -46.493,E3 +26957.243,E4 +0.000} C_DIS
LIN {X -190.174,Y +1086.028,Z +0.000,A -0.000,E1 -46.483,E3 +26966.137,E4 +0.000} C_DIS
LIN {X -190.200,Y +1096.186,Z +0.000,A -0.000,E1 -46.448,E3 +26979.141,E4 +0.000} C_DIS
LIN {X -190.154,Y +1108.998,Z +0.000,A -0.054,E1 -46.295,E3 +26995.636,E4 +0.000} C_DIS
LIN {X -189.772,Y +1119.341,Z +0.000,A -0.752,E1 -45.902,E3 +27009.174,E4 +0.000} C_DIS
LIN {X -189.097,Y +1124.276,Z +0.000,A -2.508,E1 -45.397,E3 +27015.906,E4 +0.000} C_DIS
LIN {X -187.410,Y +1129.069,Z +0.000,A -5.304,E1 -44.585,E3 +27023.079,E4 +0.000} C_DIS
LIN {X -183.899,Y +1134.873,Z +0.000,A -10.372,E1 -42.805,E3 +27033.085,E4 +0.000} C_DIS
LIN {X -179.711,Y +1140.065,Z +0.000,A -15.940,E1 -40.393,E3 +27043.871,E4 +0.000} C_DIS
LIN {X -176.763,Y +1143.197,Z +0.000,A -18.748,E1 -38.674,E3 +27051.609,E4 +0.000} C_DIS
LIN {X -172.185,Y +1147.423,Z +0.000,A -19.971,E1 -36.175,E3 +27064.339,E4 +0.000} C_DIS
LIN {X -165.999,Y +1152.127,Z +0.000,A -20.000,E1 -32.027,E3 +27084.097,E4 +0.000} C_DIS
LIN {X -160.138,Y +1155.667,Z +0.000,A -20.000,E1 -26.368,E3 +27108.467,E4 +0.000} C_DIS
LIN {X -155.625,Y +1157.756,Z +0.000,A -20.000,E1 -19.505,E3 +27137.143,E4 +0.000} C_DIS
LIN {X -153.552,Y +1158.113,Z +0.000,A -20.000,E1 -11.113,E3 +27172.894,E4 +0.000} C_DIS
LIN {X -156.311,Y +1155.540,Z +0.000,A -20.000,E1 -0.839,E3 +27216.254,E4 +0.000} C_DIS
LIN {X -161.281,Y +1151.851,Z +0.000,A -20.000,E1 +7.737,E3 +27246.153,E4 +0.000} C_DIS
LIN {X -167.493,Y +1147.157,Z +0.000,A -20.000,E1 +16.195,E3 +27270.592,E4 +0.000} C_DIS
LIN {X -173.235,Y +1142.221,Z +0.000,A -20.000,E1 +22.930,E3 +27287.894,E4 +0.000} C_DIS
LIN {X -181.123,Y +1133.734,Z +0.000,A -20.000,E1 +30.868,E3 +27308.650,E4 +0.000} C_DIS
LIN {X -189.654,Y +1120.856,Z +0.000,A -20.000,E1 +39.018,E3 +27330.664,E4 +0.000} C_DIS
LIN {X -195.246,Y +1107.046,Z +0.000,A -20.000,E1 +44.515,E3 +27348.566,E4 +0.000} C_DIS
LIN {X -198.051,Y +1092.368,Z +0.000,A -20.000,E1 +47.947,E3 +27365.092,E4 +0.000} C_DIS
LIN {X -198.143,Y +1081.370,Z +0.000,A -19.806,E1 +49.153,E3 +27376.953,E4 +0.000} C_DIS
LIN {X -197.177,Y +1073.569,Z +0.000,A -17.356,E1 +49.162,E3 +27385.537,E4 +0.000} C_DIS
LIN {X -195.448,Y +1066.139,Z +0.000,A -12.154,E1 +48.512,E3 +27394.132,E4 +0.000} C_DIS
LIN {X -193.346,Y +1058.941,Z +0.000,A -7.133,E1 +47.724,E3 +27403.012,E4 +0.000} C_DIS
LIN {X -191.781,Y +1050.839,Z +0.000,A -3.715,E1 +47.274,E3 +27413.345,E4 +0.000} C_DIS
LIN {X -190.795,Y +1039.355,Z +0.000,A -0.983,E1 +46.842,E3 +27428.005,E4 +0.000} C_DIS
LIN {X -190.395,Y +1028.856,Z +0.000,A -0.089,E1 +46.598,E3 +27441.399,E4 +0.000} C_DIS
LIN {X -190.239,Y +1018.851,Z +0.000,A -0.004,E1 +46.529,E3 +27454.167,E4 +0.000} C_DIS
LIN {X -190.161,Y +1004.975,Z +0.000,A +0.000,E1 +46.506,E3 +27471.881,E4 +0.000} C_DIS
LIN {X -190.142,Y +412.853,Z +0.000,A +0.000,E1 +46.501,E3 +28228.087,E4 +0.000} C_DIS
LIN {X -190.147,Y +401.077,Z +0.000,A +0.000,E1 +46.499,E3 +28243.128,E4 +0.000} C_DIS
LIN {X -190.159,Y +390.929,Z +0.000,A +0.000,E1 +46.494,E3 +28256.094,E4 +0.000} C_DIS
LIN {X -190.174,Y +383.973,Z +0.000,A +0.000,E1 +46.484,E3 +28264.987,E4 +0.000} C_DIS
LIN {X -190.200,Y +373.815,Z +0.000,A +0.000,E1 +46.448,E3 +28277.992,E4 +0.000} C_DIS
LIN {X -190.154,Y +361.003,Z +0.000,A +0.000,E1 +46.303,E3 +28294.486,E4 +0.000} C_DIS
LIN {X -189.772,Y +350.660,Z +0.000,A +0.049,E1 +45.996,E3 +28308.025,E4 +0.000} C_DIS
LIN {X -189.325,Y +346.917,Z +0.000,A +0.243,E1 +45.771,E3 +28313.094,E4 +0.000} C_DIS
LIN {X -188.196,Y +342.754,Z +0.000,A +1.966,E1 +45.249,E3 +28319.102,E4 +0.000} C_DIS
LIN {X -185.199,Y +337.023,Z +0.000,A +6.630,E1 +43.793,E3 +28328.476,E4 +0.000} C_DIS
LIN {X -181.141,Y +331.596,Z +0.000,A +12.274,E1 +41.569,E3 +28339.036,E4 +0.000} C_DIS
LIN {X -176.762,Y +326.804,Z +0.000,A +17.560,E1 +38.898,E3 +28350.460,E4 +0.000} C_DIS
LIN {X -172.184,Y +322.578,Z +0.000,A +19.859,E1 +36.197,E3 +28363.190,E4 +0.000} C_DIS
LIN {X -165.998,Y +317.874,Z +0.000,A +20.000,E1 +32.027,E3 +28382.948,E4 +0.000} C_DIS
LIN {X -160.137,Y +314.334,Z +0.000,A +20.000,E1 +26.368,E3 +28407.317,E4 +0.000} C_DIS
LIN {X -155.624,Y +312.245,Z +0.000,A +20.000,E1 +19.506,E3 +28435.993,E4 +0.000} C_DIS
LIN {X -153.557,Y +311.879,Z +0.000,A +20.000,E1 +11.113,E3 +28471.748,E4 +0.000} C_DIS
LIN {X -155.320,Y +313.348,Z +0.000,A +20.000,E1 +3.401,E3 +28504.932,E4 +0.000} C_DIS
LIN {X -160.005,Y +315.804,Z +0.000,A +20.000,E1 -4.720,E3 +28535.310,E4 +0.000} C_DIS
LIN {X -164.504,Y +318.255,Z +0.000,A +20.000,E1 -10.663,E3 +28554.679,E4 +0.000} C_DIS
LIN {X -170.340,Y +322.684,Z +0.000,A +20.000,E1 -17.457,E3 +28574.711,E4 +0.000} C_DIS
LIN {X -175.568,Y +329.106,Z +0.000,A +20.000,E1 -24.747,E3 +28591.945,E4 +0.000} C_DIS
LIN {X -184.074,Y +340.065,Z +0.000,A +20.000,E1 -33.664,E3 +28614.885,E4 +0.000} C_DIS
LIN {X -190.779,Y +351.388,Z +0.000,A +20.000,E1 -40.083,E3 +28632.663,E4 +0.000} C_DIS
LIN {X -195.254,Y +362.955,Z +0.000,A +20.000,E1 -44.515,E3 +28647.416,E4 +0.000} C_DIS
LIN {X -197.754,Y +374.780,Z +0.000,A +20.000,E1 -47.450,E3 +28660.838,E4 +0.000} C_DIS
LIN {X -198.310,Y +383.215,Z +0.000,A +19.956,E1 -48.698,E3 +28669.962,E4 +0.000} C_DIS
LIN {X -197.912,Y +391.275,Z +0.000,A +18.601,E1 -49.158,E3 +28678.680,E4 +0.000} C_DIS
LIN {X -196.679,Y +398.944,Z +0.000,A +13.989,E1 -48.784,E3 +28687.234,E4 +0.000} C_DIS
LIN {X -194.742,Y +406.288,Z +0.000,A +8.476,E1 -48.001,E3 +28695.917,E4 +0.000} C_DIS
LIN {X -192.748,Y +413.472,Z +0.000,A +3.905,E1 -47.267,E3 +28704.927,E4 +0.000} C_DIS
LIN {X -191.781,Y +419.162,Z +0.000,A +1.739,E1 -46.975,E3 +28712.195,E4 +0.000} C_DIS
LIN {X -190.795,Y +430.646,Z +0.000,A +0.152,E1 -46.707,E3 +28726.856,E4 +0.000} C_DIS
LIN {X -190.395,Y +441.145,Z +0.000,A +0.001,E1 -46.583,E3 +28740.249,E4 +0.000} C_DIS
LIN {X -190.239,Y +451.150,Z +0.000,A -0.000,E1 -46.528,E3 +28753.017,E4 +0.000} C_DIS
LIN {X -190.161,Y +465.026,Z +0.000,A -0.000,E1 -46.506,E3 +28770.732,E4 +0.000} C_DIS
LIN {X -190.142,Y +1057.148,Z +0.000,A -0.000,E1 -46.500,E3 +29526.938,E4 +0.000} C_DIS
LIN {X -190.147,Y +1068.924,Z +0.000,A -0.000,E1 -46.499,E3 +29541.979,E4 +0.000} C_DIS
LIN {X -190.159,Y +1079.072,Z +0.000,A -0.000,E1 -46.493,E3 +29554.944,E4 +0.000} C_DIS
LIN {X -190.174,Y +1086.028,Z +0.000,A -0.000,E1 -46.483,E3 +29563.838,E4 +0.000} C_DIS
LIN {X -190.200,Y +1096.186,Z +0.000,A -0.000,E1 -46.448,E3 +29576.842,E4 +0.000} C_DIS
LIN {X -190.154,Y +1108.998,Z +0.000,A -0.054,E1 -46.295,E3 +29593.337,E4 +0.000} C_DIS
LIN {X -189.772,Y +1119.341,Z +0.000,A -0.752,E1 -45.902,E3 +29606.875,E4 +0.000} C_DIS
LIN {X -189.097,Y +1124.276,Z +0.000,A -2.508,E1 -45.397,E3 +29613.607,E4 +0.000} C_DIS
LIN {X -187.410,Y +1129.069,Z +0.000,A -5.304,E1 -44.585,E3 +29620.780,E4 +0.000} C_DIS
LIN {X -183.899,Y +1134.873,Z +0.000,A -10.372,E1 -42.805,E3 +29630.786,E4 +0.000} C_DIS
LIN {X -179.711,Y +1140.065,Z +0.000,A -15.940,E1 -40.393,E3 +29641.572,E4 +0.000} C_DIS
LIN {X -176.763,Y +1143.197,Z +0.000,A -18.748,E1 -38.674,E3 +29649.310,E4 +0.000} C_DIS
LIN {X -172.185,Y +1147.423,Z +0.000,A -19.971,E1 -36.175,E3 +29662.040,E4 +0.000} C_DIS
LIN {X -165.999,Y +1152.127,Z +0.000,A -20.000,E1 -32.027,E3 +29681.798,E4 +0.000} C_DIS
LIN {X -160.138,Y +1155.667,Z +0.000,A -20.000,E1 -26.368,E3 +29706.168,E4 +0.000} C_DIS
LIN {X -155.625,Y +1157.756,Z +0.000,A -20.000,E1 -19.505,E3 +29734.844,E4 +0.000} C_DIS
LIN {X -153.552,Y +1158.113,Z +0.000,A -20.000,E1 -11.113,E3 +29770.595,E4 +0.000} C_DIS
LIN {X -156.311,Y +1155.540,Z +0.000,A -20.000,E1 -0.839,E3 +29813.955,E4 +0.000} C_DIS
LIN {X -161.281,Y +1151.851,Z +0.000,A -20.000,E1 +7.737,E3 +29843.854,E4 +0.000} C_DIS
LIN {X -167.493,Y +1147.157,Z +0.000,A -20.000,E1 +16.195,E3 +29868.293,E4 +0.000} C_DIS
LIN {X -173.235,Y +1142.221,Z +0.000,A -20.000,E1 +22.930,E3 +29885.595,E4 +0.000} C_DIS
LIN {X -181.123,Y +1133.734,Z +0.000,A -20.000,E1 +30.868,E3 +29906.351,E4 +0.000} C_DIS
LIN {X -189.654,Y +1120.856,Z +0.000,A -20.000,E1 +39.018,E3 +29928.365,E4 +0.000} C_DIS
LIN {X -195.246,Y +1107.046,Z +0.000,A -20.000,E1 +44.515,E3 +29946.267,E4 +0.000} C_DIS
LIN {X -198.051,Y +1092.368,Z +0.000,A -20.000,E1 +47.947,E3 +29962.793,E4 +0.000} C_DIS
LIN {X -198.143,Y +1081.370,Z +0.000,A -19.806,E1 +49.153,E3 +29974.654,E4 +0.000} C_DIS
LIN {X -197.177,Y +1073.569,Z +0.000,A -17.356,E1 +49.162,E3 +29983.238,E4 +0.000} C_DIS
LIN {X -195.448,Y +1066.139,Z +0.000,A -12.154,E1 +48.512,E3 +29991.833,E4 +0.000} C_DIS
LIN {X -193.346,Y +1058.941,Z +0.000,A -7.133,E1 +47.724,E3 +30000.713,E4 +0.000} C_DIS
LIN {X -191.781,Y +1050.839,Z +0.000,A -3.715,E1 +47.274,E3 +30011.046,E4 +0.000} C_DIS
LIN {X -190.795,Y +1039.355,Z +0.000,A -0.983,E1 +46.842,E3 +30025.706,E4 +0.000} C_DIS
LIN {X -190.395,Y +1028.856,Z +0.000,A -0.089,E1 +46.598,E3 +30039.100,E4 +0.000} C_DIS
LIN {X -190.239,Y +1018.851,Z +0.000,A -0.004,E1 +46.529,E3 +30051.868,E4 +0.000} C_DIS
LIN {X -190.161,Y +1004.975,Z +0.000,A +0.000,E1 +46.506,E3 +30069.582,E4 +0.000} C_DIS
LIN {X -190.142,Y +412.853,Z +0.000,A +0.000,E1 +46.501,E3 +30825.788,E4 +0.000} C_DIS
LIN {X -190.147,Y +401.077,Z +0.000,A +0.000,E1 +46.499,E3 +30840.829,E4 +0.000} C_DIS
LIN {X -190.159,Y +390.929,Z +0.000,A +0.000,E1 +46.494,E3 +30853.795,E4 +0.000} C_DIS
LIN {X -190.174,Y +383.973,Z +0.000,A +0.000,E1 +46.484,E3 +30862.688,E4 +0.000} C_DIS
LIN {X -190.200,Y +373.815,Z +0.000,A +0.000,E1 +46.448,E3 +30875.693,E4 +0.000} C_DIS
LIN {X -190.154,Y +361.003,Z +0.000,A +0.000,E1 +46.303,E3 +30892.187,E4 +0.000} C_DIS
LIN {X -189.772,Y +350.660,Z +0.000,A +0.049,E1 +45.996,E3 +30905.726,E4 +0.000} C_DIS
LIN {X -189.325,Y +346.917,Z +0.000,A +0.243,E1 +45.771,E3 +30910.795,E4 +0.000} C_DIS
LIN {X -188.196,Y +342.754,Z +0.000,A +1.966,E1 +45.249,E3 +30916.803,E4 +0.000} C_DIS
LIN {X -185.199,Y +337.023,Z +0.000,A +6.630,E1 +43.793,E3 +30926.177,E4 +0.000} C_DIS
LIN {X -181.141,Y +331.596,Z +0.000,A +12.274,E1 +41.569,E3 +30936.737,E4 +0.000} C_DIS
LIN {X -176.762,Y +326.804,Z +0.000,A +17.560,E1 +38.898,E3 +30948.161,E4 +0.000} C_DIS
LIN {X -172.184,Y +322.578,Z +0.000,A +19.859,E1 +36.197,E3 +30960.891,E4 +0.000} C_DIS
LIN {X -165.998,Y +317.874,Z +0.000,A +20.000,E1 +32.027,E3 +30980.649,E4 +0.000} C_DIS
LIN {X -160.137,Y +314.334,Z +0.000,A +20.000,E1 +26.368,E3 +31005.018,E4 +0.000} C_DIS
LIN {X -155.624,Y +312.245,Z +0.000,A +20.000,E1 +19.506,E3 +31033.694,E4 +0.000} C_DIS
LIN {X -153.557,Y +311.879,Z +0.000,A +20.000,E1 +11.113,E3 +31069.449,E4 +0.000} C_DIS
LIN {X -155.320,Y +313.348,Z +0.000,A +20.000,E1 +3.401,E3 +31102.633,E4 +0.000} C_DIS
LIN {X -160.005,Y +315.804,Z +0.000,A +20.000,E1 -4.720,E3 +31133.011,E4 +0.000} C_DIS
LIN {X -164.504,Y +318.255,Z +0.000,A +20.000,E1 -10.663,E3 +31152.380,E4 +0.000} C_DIS
LIN {X -170.340,Y +322.684,Z +0.000,A +20.000,E1 -17.457,E3 +31172.412,E4 +0.000} C_DIS
LIN {X -175.568,Y +329.106,Z +0.000,A +20.000,E1 -24.747,E3 +31189.646,E4 +0.000} C_DIS
LIN {X -184.074,Y +340.065,Z +0.000,A +20.000,E1 -33.664,E3 +31212.586,E4 +0.000} C_DIS
LIN {X -190.779,Y +351.388,Z +0.000,A +20.000,E1 -40.083,E3 +31230.364,E4 +0.000} C_DIS
LIN {X -195.254,Y +362.955,Z +0.000,A +20.000,E1 -44.515,E3 +31245.117,E4 +0.000} C_DIS
LIN {X -197.754,Y +374.780,Z +0.000,A +20.000,E1 -47.450,E3 +31258.539,E4 +0.000} C_DIS
LIN {X -198.310,Y +383.215,Z +0.000,A +19.956,E1 -48.698,E3 +31267.663,E4 +0.000} C_DIS
LIN {X -197.912,Y +391.275,Z +0.000,A +18.601,E1 -49.158,E3 +31276.381,E4 +0.000} C_DIS
LIN {X -196.679,Y +398.944,Z +0.000,A +13.989,E1 -48.784,E3 +31284.935,E4 +0.000} C_DIS
LIN {X -194.742,Y +406.288,Z +0.000,A +8.476,E1 -48.001,E3 +31293.618,E4 +0.000} C_DIS
LIN {X -192.748,Y +413.472,Z +0.000,A +3.905,E1 -47.267,E3 +31302.628,E4 +0.000} C_DIS
LIN {X -191.781,Y +419.162,Z +0.000,A +1.739,E1 -46.975,E3 +31309.896,E4 +0.000} C_DIS
LIN {X -190.795,Y +430.646,Z +0.000,A +0.152,E1 -46.707,E3 +31324.557,E4 +0.000} C_DIS
LIN {X -190.395,Y +441.145,Z +0.000,A +0.001,E1 -46.583,E3 +31337.950,E4 +0.000} C_DIS
LIN {X -190.239,Y +451.150,Z +0.000,A -0.000,E1 -46.528,E3 +31350.718,E4 +0.000} C_DIS
LIN {X -190.161,Y +465.026,Z +0.000,A -0.000,E1 -46.506,E3 +31368.433,E4 +0.000} C_DIS
LIN {X -190.142,Y +1057.148,Z +0.000,A -0.000,E1 -46.500,E3 +32124.639,E4 +0.000} C_DIS
LIN {X -190.147,Y +1068.924,Z +0.000,A -0.000,E1 -46.499,E3 +32139.680,E4 +0.000} C_DIS
LIN {X -190.159,Y +1079.072,Z +0.000,A -0.000,E1 -46.493,E3 +32152.645,E4 +0.000} C_DIS
LIN {X -190.174,Y +1086.028,Z +0.000,A -0.000,E1 -46.483,E3 +32161.539,E4 +0.000} C_DIS
LIN {X -190.200,Y +1096.186,Z +0.000,A -0.000,E1 -46.448,E3 +32174.543,E4 +0.000} C_DIS
LIN {X -190.154,Y +1108.998,Z +0.000,A -0.054,E1 -46.295,E3 +32191.038,E4 +0.000} C_DIS
LIN {X -189.772,Y +1119.341,Z +0.000,A -0.752,E1 -45.902,E3 +32204.576,E4 +0.000} C_DIS
LIN {X -189.097,Y +1124.276,Z +0.000,A -2.508,E1 -45.397,E3 +32211.308,E4 +0.000} C_DIS
LIN {X -187.410,Y +1129.069,Z +0.000,A -5.304,E1 -44.585,E3 +32218.481,E4 +0.000} C_DIS
LIN {X -183.899,Y +1134.873,Z +0.000,A -10.372,E1 -42.805,E3 +32228.487,E4 +0.000} C_DIS
LIN {X -179.711,Y +1140.065,Z +0.000,A -15.940,E1 -40.393,E3 +32239.273,E4 +0.000} C_DIS
LIN {X -176.763,Y +1143.197,Z +0.000,A -18.748,E1 -38.674,E3 +32247.011,E4 +0.000} C_DIS
LIN {X -172.185,Y +1147.423,Z +0.000,A -19.971,E1 -36.175,E3 +32259.741,E4 +0.000} C_DIS
LIN {X -165.999,Y +1152.127,Z +0.000,A -20.000,E1 -32.027,E3 +32279.499,E4 +0.000} C_DIS
LIN {X -160.138,Y +1155.667,Z +0.000,A -20.000,E1 -26.368,E3 +32303.869,E4 +0.000} C_DIS
LIN {X -155.625,Y +1157.756,Z +0.000,A -20.000,E1 -19.505,E3 +32332.545,E4 +0.000} C_DIS
LIN {X -153.552,Y +1158.113,Z +0.000,A -20.000,E1 -11.113,E3 +32368.296,E4 +0.000} C_DIS
LIN {X -156.311,Y +1155.540,Z +0.000,A -20.000,E1 -0.839,E3 +32411.656,E4 +0.000} C_DIS
LIN {X -161.281,Y +1151.851,Z +0.000,A -20.000,E1 +7.737,E3 +32441.555,E4 +0.000} C_DIS
LIN {X -167.493,Y +1147.157,Z +0.000,A -20.000,E1 +16.195,E3 +32465.994,E4 +0.000} C_DIS
LIN {X -173.235,Y +1142.221,Z +0.000,A -20.000,E1 +22.930,E3 +32483.296,E4 +0.000} C_DIS
LIN {X -181.123,Y +1133.734,Z +0.000,A -20.000,E1 +30.868,E3 +32504.052,E4 +0.000} C_DIS
LIN {X -189.654,Y +1120.856,Z +0.000,A -20.000,E1 +39.018,E3 +32526.066,E4 +0.000} C_DIS
LIN {X -195.246,Y +1107.046,Z +0.000,A -20.000,E1 +44.515,E3 +32543.968,E4 +0.000} C_DIS
LIN {X -198.051,Y +1092.368,Z +0.000,A -20.000,E1 +47.947,E3 +32560.494,E4 +0.000} C_DIS
LIN {X -198.143,Y +1081.370,Z +0.000,A -19.806,E1 +49.153,E3 +32572.355,E4 +0.000} C_DIS
LIN {X -197.177,Y +1073.569,Z +0.000,A -17.356,E1 +49.162,E3 +32580.939,E4 +0.000} C_DIS
LIN {X -195.448,Y +1066.139,Z +0.000,A -12.154,E1 +48.512,E3 +32589.534,E4 +0.000} C_DIS
LIN {X -193.346,Y +1058.941,Z +0.000,A -7.133,E1 +47.724,E3 +32598.414,E4 +0.000} C_DIS
LIN {X -191.781,Y +1050.839,Z +0.000,A -3.715,E1 +47.274,E3 +32608.747,E4 +0.000} C_DIS
LIN {X -190.795,Y +1039.355,Z +0.000,A -0.983,E1 +46.842,E3 +32623.407,E4 +0.000} C_DIS
LIN {X -190.395,Y +1028.856,Z +0.000,A -0.089,E1 +46.598,E3 +32636.801,E4 +0.000} C_DIS
LIN {X -190.239,Y +1018.851,Z +0.000,A -0.004,E1 +46.529,E3 +32649.569,E4 +0.000} C_DIS
LIN {X -190.161,Y +1004.975,Z +0.000,A +0.000,E1 +46.506,E3 +32667.283,E4 +0.000} C_DIS
LIN {X -190.142,Y +412.853,Z +0.000,A +0.000,E1 +46.501,E3 +33423.489,E4 +0.000} C_DIS
LIN {X -190.147,Y +401.077,Z +0.000,A +0.000,E1 +46.499,E3 +33438.530,E4 +0.000} C_DIS
LIN {X -190.159,Y +390.929,Z +0.000,A +0.000,E1 +46.494,E3 +33451.496,E4 +0.000} C_DIS
LIN {X -190.174,Y +383.973,Z +0.000,A +0.000,E1 +46.484,E3 +33460.389,E4 +0.000} C_DIS
LIN {X -190.200,Y +373.815,Z +0.000,A +0.000,E1 +46.448,E3 +33473.394,E4 +0.000} C_DIS
LIN {X -190.154,Y +361.003,Z +0.000,A +0.000,E1 +46.303,E3 +33489.888,E4 +0.000} C_DIS
LIN {X -189.772,Y +350.660,Z +0.000,A +0.049,E1 +45.996,E3 +33503.427,E4 +0.000} C_DIS
LIN {X -189.325,Y +346.917,Z +0.000,A +0.243,E1 +45.771,E3 +33508.496,E4 +0.000} C_DIS
LIN {X -188.196,Y +342.754,Z +0.000,A +1.966,E1 +45.249,E3 +33514.504,E4 +0.000} C_DIS
LIN {X -185.199,Y +337.023,Z +0.000,A +6.630,E1 +43.793,E3 +33523.878,E4 +0.000} C_DIS
LIN {X -181.141,Y +331.596,Z +0.000,A +12.274,E1 +41.569,E3 +33534.438,E4 +0.000} C_DIS
LIN {X -176.762,Y +326.804,Z +0.000,A +17.560,E1 +38.898,E3 +33545.862,E4 +0.000} C_DIS
LIN {X -172.184,Y +322.578,Z +0.000,A +19.859,E1 +36.197,E3 +33558.592,E4 +0.000} C_DIS
LIN {X -165.998,Y +317.874,Z +0.000,A +20.000,E1 +32.027,E3 +33578.350,E4 +0.000} C_DIS
LIN {X -160.137,Y +314.334,Z +0.000,A +20.000,E1 +26.368,E3 +33602.719,E4 +0.000} C_DIS
LIN {X -155.624,Y +312.245,Z +0.000,A +20.000,E1 +19.506,E3 +33631.395,E4 +0.000} C_DIS
LIN {X -153.557,Y +311.879,Z +0.000,A +20.000,E1 +11.113,E3 +33667.150,E4 +0.000} C_DIS
LIN {X -155.320,Y +313.348,Z +0.000,A +20.000,E1 +3.401,E3 +33700.334,E4 +0.000} C_DIS
LIN {X -160.005,Y +315.804,Z +0.000,A +20.000,E1 -4.720,E3 +33730.712,E4 +0.000} C_DIS
LIN {X -164.504,Y +318.255,Z +0.000,A +20.000,E1 -10.663,E3 +33750.081,E4 +0.000} C_DIS
LIN {X -170.340,Y +322.684,Z +0.000,A +20.000,E1 -17.457,E3 +33770.113,E4 +0.000} C_DIS
LIN {X -175.568,Y +329.106,Z +0.000,A +20.000,E1 -24.747,E3 +33787.347,E4 +0.000} C_DIS
LIN {X -184.074,Y +340.065,Z +0.000,A +20.000,E1 -33.664,E3 +33810.287,E4 +0.000} C_DIS
LIN {X -190.779,Y +351.388,Z +0.000,A +20.000,E1 -40.083,E3 +33828.065,E4 +0.000} C_DIS
LIN {X -195.254,Y +362.955,Z +0.000,A +20.000,E1 -44.515,E3 +33842.818,E4 +0.000} C_DIS
LIN {X -197.754,Y +374.780,Z +0.000,A +20.000,E1 -47.450,E3 +33856.240,E4 +0.000} C_DIS
LIN {X -198.310,Y +383.215,Z +0.000,A +19.956,E1 -48.698,E3 +33865.364,E4 +0.000} C_DIS
LIN {X -197.912,Y +391.275,Z +0.000,A +18.601,E1 -49.158,E3 +33874.082,E4 +0.000} C_DIS
LIN {X -196.679,Y +398.944,Z +0.000,A +13.989,E1 -48.784,E3 +33882.636,E4 +0.000} C_DIS
LIN {X -194.742,Y +406.288,Z +0.000,A +8.476,E1 -48.001,E3 +33891.319,E4 +0.000} C_DIS
LIN {X -192.748,Y +413.472,Z +0.000,A +3.905,E1 -47.267,E3 +33900.329,E4 +0.000} C_DIS
LIN {X -191.781,Y +419.162,Z +0.000,A +1.739,E1 -46.975,E3 +33907.597,E4 +0.000} C_DIS
LIN {X -190.795,Y +430.646,Z +0.000,A +0.152,E1 -46.707,E3 +33922.258,E4 +0.000} C_DIS
LIN {X -190.395,Y +441.145,Z +0.000,A +0.001,E1 -46.583,E3 +33935.651,E4 +0.000} C_DIS
LIN {X -190.239,Y +451.150,Z +0.000,A -0.000,E1 -46.528,E3 +33948.419,E4 +0.000} C_DIS
LIN {X -190.161,Y +465.026,Z +0.000,A -0.000,E1 -46.506,E3 +33966.134,E4 +0.000} C_DIS
LIN {X -190.142,Y +1057.148,Z +0.000,A -0.000,E1 -46.500,E3 +34722.340,E4 +0.000} C_DIS
LIN {X -190.147,Y +1068.924,Z +0.000,A -0.000,E1 -46.499,E3 +34737.381,E4 +0.000} C_DIS
LIN {X -190.159,Y +1079.072,Z +0.000,A -0.000,E1 -46.493,E3 +34750.346,E4 +0.000} C_DIS
LIN {X -190.174,Y +1086.028,Z +0.000,A -0.000,E1 -46.483,E3 +34759.240,E4 +0.000} C_DIS
LIN {X -190.200,Y +1096.186,Z +0.000,A -0.000,E1 -46.448,E3 +34772.244,E4 +0.000} C_DIS
LIN {X -190.154,Y +1108.998,Z +0.000,A -0.054,E1 -46.295,E3 +34788.739,E4 +0.000} C_DIS
LIN {X -189.772,Y +1119.341,Z +0.000,A -0.752,E1 -45.902,E3 +34802.277,E4 +0.000} C_DIS
LIN {X -189.097,Y +1124.276,Z +0.000,A -2.508,E1 -45.397,E3 +34809.009,E4 +0.000} C_DIS
LIN {X -187.410,Y +1129.069,Z +0.000,A -5.304,E1 -44.585,E3 +34816.182,E4 +0.000} C_DIS
LIN {X -183.899,Y +1134.873,Z +0.000,A -10.372,E1 -42.805,E3 +34826.188,E4 +0.000} C_DIS
LIN {X -179.711,Y +1140.065,Z +0.000,A -15.940,E1 -40.393,E3 +34836.974,E4 +0.000} C_DIS
LIN {X -176.763,Y +1143.197,Z +0.000,A -18.748,E1 -38.674,E3 +34844.712,E4 +0.000} C_DIS
LIN {X -172.185,Y +1147.423,Z +0.000,A -19.971,E1 -36.175,E3 +34857.442,E4 +0.000} C_DIS
LIN {X -165.999,Y +1152.127,Z +0.000,A -20.000,E1 -32.027,E3 +34877.200,E4 +0.000} C_DIS
LIN {X -160.138,Y +1155.667,Z +0.000,A -20.000,E1 -26.368,E3 +34901.570,E4 +0.000} C_DIS
LIN {X -155.625,Y +1157.756,Z +0.000,A -20.000,E1 -19.505,E3 +34930.246,E4 +0.000} C_DIS
LIN {X -153.552,Y +1158.113,Z +0.000,A -20.000,E1 -11.113,E3 +34965.997,E4 +0.000} C_DIS
LIN {X -156.311,Y +1155.540,Z +0.000,A -20.000,E1 -0.839,E3 +35009.357,E4 +0.000} C_DIS
LIN {X -161.281,Y +1151.851,Z +0.000,A -20.000,E1 +7.737,E3 +35039.256,E4 +0.000} C_DIS
LIN {X -167.493,Y +1147.157,Z +0.000,A -20.000,E1 +16.195,E3 +35063.695,E4 +0.000} C_DIS
LIN {X -173.235,Y +1142.221,Z +0.000,A -20.000,E1 +22.930,E3 +35080.997,E4 +0.000} C_DIS
LIN {X -181.123,Y +1133.734,Z +0.000,A -20.000,E1 +30.868,E3 +35101.753,E4 +0.000} C_DIS
LIN {X -189.654,Y +1120.856,Z +0.000,A -20.000,E1 +39.018,E3 +35123.767,E4 +0.000} C_DIS
LIN {X -195.246,Y +1107.046,Z +0.000,A -20.000,E1 +44.515,E3 +35141.669,E4 +0.000} C_DIS
LIN {X -198.051,Y +1092.368,Z +0.000,A -20.000,E1 +47.947,E3 +35158.195,E4 +0.000} C_DIS
LIN {X -198.143,Y +1081.370,Z +0.000,A -19.806,E1 +49.153,E3 +35170.056,E4 +0.000} C_DIS
LIN {X -197.177,Y +1073.569,Z +0.000,A -17.356,E1 +49.162,E3 +35178.640,E4 +0.000} C_DIS
LIN {X -195.448,Y +1066.139,Z +0.000,A -12.154,E1 +48.512,E3 +35187.235,E4 +0.000} C_DIS
LIN {X -193.346,Y +1058.941,Z +0.000,A -7.133,E1 +47.724,E3 +35196.115,E4 +0.000} C_DIS
LIN {X -191.781,Y +1050.839,Z +0.000,A -3.715,E1 +47.274,E3 +35206.448,E4 +0.000} C_DIS
LIN {X -190.795,Y +1039.355,Z +0.000,A -0.983,E1 +46.842,E3 +35221.108,E4 +0.000} C_DIS
LIN {X -190.395,Y +1028.856,Z +0.000,A -0.089,E1 +46.598,E3 +35234.502,E4 +0.000} C_DIS
LIN {X -190.239,Y +1018.851,Z +0.000,A -0.004,E1 +46.529,E3 +35247.270,E4 +0.000} C_DIS
LIN {X -190.161,Y +1004.975,Z +0.000,A +0.000,E1 +46.506,E3 +35264.984,E4 +0.000} C_DIS
LIN {X -190.142,Y +412.853,Z +0.000,A +0.000,E1 +46.501,E3 +36021.190,E4 +0.000} C_DIS
LIN {X -190.147,Y +401.077,Z +0.000,A +0.000,E1 +46.499,E3 +36036.231,E4 +0.000} C_DIS
LIN {X -190.159,Y +390.929,Z +0.000,A +0.000,E1 +46.494,E3 +36049.197,E4 +0.000} C_DIS
LIN {X -190.174,Y +383.973,Z +0.000,A +0.000,E1 +46.484,E3 +36058.090,E4 +0.000} C_DIS
LIN {X -190.200,Y +373.815,Z +0.000,A +0.000,E1 +46.448,E3 +36071.095,E4 +0.000} C_DIS
LIN {X -190.154,Y +361.003,Z +0.000,A +0.000,E1 +46.303,E3 +36087.589,E4 +0.000} C_DIS
LIN {X -189.772,Y +350.660,Z +0.000,A +0.049,E1 +45.996,E3 +36101.128,E4 +0.000} C_DIS
LIN {X -189.325,Y +346.917,Z +0.000,A +0.243,E1 +45.771,E3 +36106.197,E4 +0.000} C_DIS
LIN {X -188.196,Y +342.754,Z +0.000,A +1.966,E1 +45.249,E3 +36112.205,E4 +0.000} C_DIS
LIN {X -185.199,Y +337.023,Z +0.000,A +6.630,E1 +43.793,E3 +36121.579,E4 +0.000} C_DIS
LIN {X -181.141,Y +331.596,Z +0.000,A +12.274,E1 +41.569,E3 +36132.139,E4 +0.000} C_DIS
LIN {X -176.762,Y +326.804,Z +0.000,A +17.560,E1 +38.898,E3 +36143.563,E4 +0.000} C_DIS
LIN {X -172.184,Y +322.578,Z +0.000,A +19.859,E1 +36.197,E3 +36156.293,E4 +0.000} C_DIS
LIN {X -165.998,Y +317.874,Z +0.000,A +20.000,E1 +32.027,E3 +36176.051,E4 +0.000} C_DIS
LIN {X -160.137,Y +314.334,Z +0.000,A +20.000,E1 +26.368,E3 +36200.420,E4 +0.000} C_DIS
LIN {X -155.624,Y +312.245,Z +0.000,A +20.000,E1 +19.506,E3 +36229.096,E4 +0.000} C_DIS
LIN {X -153.557,Y +311.879,Z +0.000,A +20.000,E1 +11.113,E3 +36264.851,E4 +0.000} C_DIS
LIN {X -155.320,Y +313.348,Z +0.000,A +20.000,E1 +3.401,E3 +36298.035,E4 +0.000} C_DIS
LIN {X -160.005,Y +315.804,Z +0.000,A +20.000,E1 -4.720,E3 +36328.413,E4 +0.000} C_DIS
LIN {X -164.504,Y +318.255,Z +0.000,A +20.000,E1 -10.663,E3 +36347.782,E4 +0.000} C_DIS
LIN {X -170.340,Y +322.684,Z +0.000,A +20.000,E1 -17.457,E3 +36367.814,E4 +0.000} C_DIS
LIN {X -175.568,Y +329.106,Z +0.000,A +20.000,E1 -24.747,E3 +36385.048,E4 +0.000} C_DIS
LIN {X -184.074,Y +340.065,Z +0.000,A +20.000,E1 -33.664,E3 +36407.988,E4 +0.000} C_DIS
LIN {X -190.779,Y +351.388,Z +0.000,A +20.000,E1 -40.083,E3 +36425.766,E4 +0.000} C_DIS
LIN {X -195.254,Y +362.955,Z +0.000,A +20.000,E1 -44.515,E3 +36440.519,E4 +0.000} C_DIS
LIN {X -197.754,Y +374.780,Z +0.000,A +20.000,E1 -47.450,E3 +36453.941,E4 +0.000} C_DIS
LIN {X -198.310,Y +383.215,Z +0.000,A +19.956,E1 -48.698,E3 +36463.065,E4 +0.000} C_DIS
LIN {X -197.912,Y +391.275,Z +0.000,A +18.601,E1 -49.158,E3 +36471.783,E4 +0.000} C_DIS
LIN {X -196.679,Y +398.944,Z +0.000,A +13.989,E1 -48.784,E3 +36480.337,E4 +0.000} C_DIS
LIN {X -194.742,Y +406.288,Z +0.000,A +8.476,E1 -48.001,E3 +36489.020,E4 +0.000} C_DIS
LIN {X -192.748,Y +413.472,Z +0.000,A +3.905,E1 -47.267,E3 +36498.030,E4 +0.000} C_DIS
LIN {X -191.781,Y +419.162,Z +0.000,A +1.739,E1 -46.975,E3 +36505.298,E4 +0.000} C_DIS
LIN {X -190.795,Y +430.646,Z +0.000,A +0.152,E1 -46.707,E3 +36519.959,E4 +0.000} C_DIS
LIN {X -190.395,Y +441.145,Z +0.000,A +0.001,E1 -46.583,E3 +36533.352,E4 +0.000} C_DIS
LIN {X -190.239,Y +451.150,Z +0.000,A -0.000,E1 -46.528,E3 +36546.120,E4 +0.000} C_DIS
LIN {X -190.161,Y +465.026,Z +0.000,A -0.000,E1 -46.506,E3 +36563.835,E4 +0.000} C_DIS
LIN {X -190.142,Y +1057.148,Z +0.000,A -0.000,E1 -46.500,E3 +37320.041,E4 +0.000} C_DIS
LIN {X -190.147,Y +1068.924,Z +0.000,A -0.000,E1 -46.499,E3 +37335.082,E4 +0.000} C_DIS
LIN {X -190.159,Y +1079.072,Z +0.000,A -0.000,E1 -46.493,E3 +37348.047,E4 +0.000} C_DIS
LIN {X -190.174,Y +1086.028,Z +0.000,A -0.000,E1 -46.483,E3 +37356.941,E4 +0.000} C_DIS
LIN {X -190.200,Y +1096.186,Z +0.000,A -0.000,E1 -46.448,E3 +37369.945,E4 +0.000} C_DIS
LIN {X -190.154,Y +1108.998,Z +0.000,A -0.054,E1 -46.295,E3 +37386.440,E4 +0.000} C_DIS
LIN {X -189.772,Y +1119.341,Z +0.000,A -0.752,E1 -45.902,E3 +37399.978,E4 +0.000} C_DIS
LIN {X -189.097,Y +1124.276,Z +0.000,A -2.508,E1 -45.397,E3 +37406.710,E4 +0.000} C_DIS
LIN {X -187.410,Y +1129.069,Z +0.000,A -5.304,E1 -44.585,E3 +37413.883,E4 +0.000} C_DIS
LIN {X -183.899,Y +1134.873,Z +0.000,A -10.372,E1 -42.805,E3 +37423.889,E4 +0.000} C_DIS
LIN {X -179.711,Y +1140.065,Z +0.000,A -15.940,E1 -40.393,E3 +37434.675,E4 +0.000} C_DIS
LIN {X -176.763,Y +1143.197,Z +0.000,A -18.748,E1 -38.674,E3 +37442.413,E4 +0.000} C_DIS
LIN {X -172.185,Y +1147.423,Z +0.000,A -19.971,E1 -36.175,E3 +37455.143,E4 +0.000} C_DIS
LIN {X -165.999,Y +1152.127,Z +0.000,A -20.000,E1 -32.027,E3 +37474.901,E4 +0.000} C_DIS
LIN {X -160.138,Y +1155.667,Z +0.000,A -20.000,E1 -26.368,E3 +37499.271,E4 +0.000} C_DIS
LIN {X -155.625,Y +1157.756,Z +0.000,A -20.000,E1 -19.505,E3 +37527.947,E4 +0.000} C_DIS
LIN {X -153.552,Y +1158.113,Z +0.000,A -20.000,E1 -11.113,E3 +37563.698,E4 +0.000} C_DIS
LIN {X -156.311,Y +1155.540,Z +0.000,A -20.000,E1 -0.839,E3 +37607.058,E4 +0.000} C_DIS
LIN {X -161.281,Y +1151.851,Z +0.000,A -20.000,E1 +7.737,E3 +37636.957,E4 +0.000} C_DIS
LIN {X -167.493,Y +1147.157,Z +0.000,A -20.000,E1 +16.195,E3 +37661.396,E4 +0.000} C_DIS
LIN {X -173.235,Y +1142.221,Z +0.000,A -20.000,E1 +22.930,E3 +37678.698,E4 +0.000} C_DIS
LIN {X -181.123,Y +1133.734,Z +0.000,A -20.000,E1 +30.868,E3 +37699.454,E4 +0.000} C_DIS
LIN {X -189.654,Y +1120.856,Z +0.000,A -20.000,E1 +39.018,E3 +37721.468,E4 +0.000} C_DIS
LIN {X -195.246,Y +1107.046,Z +0.000,A -20.000,E1 +44.515,E3 +37739.370,E4 +0.000} C_DIS
LIN {X -198.051,Y +1092.368,Z +0.000,A -20.000,E1 +47.947,E3 +37755.896,E4 +0.000} C_DIS
LIN {X -198.143,Y +1081.370,Z +0.000,A -19.806,E1 +49.153,E3 +37767.757,E4 +0.000} C_DIS
LIN {X -197.177,Y +1073.569,Z +0.000,A -17.356,E1 +49.162,E3 +37776.341,E4 +0.000} C_DIS
LIN {X -195.448,Y +1066.139,Z +0.000,A -12.154,E1 +48.512,E3 +37784.936,E4 +0.000} C_DIS
LIN {X -193.346,Y +1058.941,Z +0.000,A -7.133,E1 +47.724,E3 +37793.816,E4 +0.000} C_DIS
LIN {X -191.781,Y +1050.839,Z +0.000,A -3.715,E1 +47.274,E3 +37804.149,E4 +0.000} C_DIS
LIN {X -190.795,Y +1039.355,Z +0.000,A -0.983,E1 +46.842,E3 +37818.809,E4 +0.000} C_DIS
LIN {X -190.395,Y +1028.856,Z +0.000,A -0.089,E1 +46.598,E3 +37832.203,E4 +0.000} C_DIS
LIN {X -190.239,Y +1018.851,Z +0.000,A -0.004,E1 +46.529,E3 +37844.971,E4 +0.000} C_DIS
LIN {X -190.161,Y +1004.975,Z +0.000,A +0.000,E1 +46.506,E3 +37862.685,E4 +0.000} C_DIS
LIN {X -190.142,Y +412.853,Z +0.000,A +0.000,E1 +46.501,E3 +38618.891,E4 +0.000} C_DIS
LIN {X -190.147,Y +401.077,Z +0.000,A +0.000,E1 +46.499,E3 +38633.932,E4 +0.000} C_DIS
LIN {X -190.159,Y +390.929,Z +0.000,A +0.000,E1 +46.494,E3 +38646.898,E4 +0.000} C_DIS
LIN {X -190.174,Y +383.973,Z +0.000,A +0.000,E1 +46.484,E3 +38655.791,E4 +0.000} C_DIS
LIN {X -190.200,Y +373.815,Z +0.000,A +0.000,E1 +46.448,E3 +38668.796,E4 +0.000} C_DIS
LIN {X -190.154,Y +361.003,Z +0.000,A +0.000,E1 +46.303,E3 +38685.290,E4 +0.000} C_DIS
LIN {X -189.772,Y +350.660,Z +0.000,A +0.049,E1 +45.996,E3 +38698.829,E4 +0.000} C_DIS
LIN {X -189.325,Y +346.917,Z +0.000,A +0.243,E1 +45.771,E3 +38703.898,E4 +0.000} C_DIS
LIN {X -188.196,Y +342.754,Z +0.000,A +1.966,E1 +45.249,E3 +38709.906,E4 +0.000} C_DIS
LIN {X -185.199,Y +337.023,Z +0.000,A +6.630,E1 +43.793,E3 +38719.280,E4 +0.000} C_DIS
LIN {X -181.141,Y +331.596,Z +0.000,A +12.274,E1 +41.569,E3 +38729.840,E4 +0.000} C_DIS
LIN {X -176.762,Y +326.804,Z +0.000,A +17.560,E1 +38.898,E3 +38741.264,E4 +0.000} C_DIS
LIN {X -172.184,Y +322.578,Z +0.000,A +19.859,E1 +36.197,E3 +38753.994,E4 +0.000} C_DIS
LIN {X -165.998,Y +317.874,Z +0.000,A +20.000,E1 +32.027,E3 +38773.752,E4 +0.000} C_DIS
LIN {X -160.137,Y +314.334,Z +0.000,A +20.000,E1 +26.368,E3 +38798.121,E4 +0.000} C_DIS
LIN {X -155.624,Y +312.245,Z +0.000,A +20.000,E1 +19.506,E3 +38826.797,E4 +0.000} C_DIS
LIN {X -153.557,Y +311.879,Z +0.000,A +20.000,E1 +11.113,E3 +38862.552,E4 +0.000} C_DIS
LIN {X -155.320,Y +313.348,Z +0.000,A +20.000,E1 +3.401,E3 +38895.736,E4 +0.000} C_DIS
LIN {X -160.005,Y +315.804,Z +0.000,A +20.000,E1 -4.720,E3 +38926.114,E4 +0.000} C_DIS
LIN {X -164.504,Y +318.255,Z +0.000,A +20.000,E1 -10.663,E3 +38945.483,E4 +0.000} C_DIS
LIN {X -170.340,Y +322.684,Z +0.000,A +20.000,E1 -17.457,E3 +38965.515,E4 +0.000} C_DIS
LIN {X -175.568,Y +329.106,Z +0.000,A +20.000,E1 -24.747,E3 +38982.749,E4 +0.000} C_DIS
LIN {X -184.074,Y +340.065,Z +0.000,A +20.000,E1 -33.664,E3 +39005.689,E4 +0.000} C_DIS
LIN {X -190.779,Y +351.388,Z +0.000,A +20.000,E1 -40.083,E3 +39023.467,E4 +0.000} C_DIS
LIN {X -195.254,Y +362.955,Z +0.000,A +20.000,E1 -44.515,E3 +39038.220,E4 +0.000} C_DIS
LIN {X -197.754,Y +374.780,Z +0.000,A +20.000,E1 -47.450,E3 +39051.642,E4 +0.000} C_DIS
LIN {X -198.310,Y +383.215,Z +0.000,A +19.956,E1 -48.698,E3 +39060.766,E4 +0.000} C_DIS
LIN {X -197.912,Y +391.275,Z +0.000,A +18.601,E1 -49.158,E3 +39069.484,E4 +0.000} C_DIS
LIN {X -196.679,Y +398.944,Z +0.000,A +13.989,E1 -48.784,E3 +39078.038,E4 +0.000} C_DIS
LIN {X -194.742,Y +406.288,Z +0.000,A +8.476,E1 -48.001,E3 +39086.721,E4 +0.000} C_DIS
LIN {X -192.748,Y +413.472,Z +0.000,A +3.905,E1 -47.267,E3 +39095.731,E4 +0.000} C_DIS
LIN {X -191.781,Y +419.162,Z +0.000,A +1.739,E1 -46.975,E3 +39102.999,E4 +0.000} C_DIS
LIN {X -190.795,Y +430.646,Z +0.000,A +0.152,E1 -46.707,E3 +39117.660,E4 +0.000} C_DIS
LIN {X -190.395,Y +441.145,Z +0.000,A +0.001,E1 -46.583,E3 +39131.053,E4 +0.000} C_DIS
LIN {X -190.239,Y +451.150,Z +0.000,A -0.000,E1 -46.528,E3 +39143.821,E4 +0.000} C_DIS
LIN {X -190.161,Y +465.026,Z +0.000,A -0.000,E1 -46.506,E3 +39161.536,E4 +0.000} C_DIS
LIN {X -190.142,Y +1057.148,Z +0.000,A -0.000,E1 -46.500,E3 +39917.742,E4 +0.000} C_DIS
LIN {X -190.147,Y +1068.924,Z +0.000,A -0.000,E1 -46.499,E3 +39932.783,E4 +0.000} C_DIS
LIN {X -190.159,Y +1079.072,Z +0.000,A -0.000,E1 -46.493,E3 +39945.748,E4 +0.000} C_DIS
LIN {X -190.174,Y +1086.028,Z +0.000,A -0.000,E1 -46.483,E3 +39954.642,E4 +0.000} C_DIS
LIN {X -190.200,Y +1096.186,Z +0.000,A -0.000,E1 -46.448,E3 +39967.646,E4 +0.000} C_DIS
LIN {X -190.154,Y +1108.998,Z +0.000,A -0.054,E1 -46.295,E3 +39984.141,E4 +0.000} C_DIS
LIN {X -189.772,Y +1119.341,Z +0.000,A -0.752,E1 -45.902,E3 +39997.679,E4 +0.000} C_DIS
LIN {X -189.097,Y +1124.276,Z +0.000,A -2.508,E1 -45.397,E3 +40004.411,E4 +0.000} C_DIS
LIN {X -187.410,Y +1129.069,Z +0.000,A -5.304,E1 -44.585,E3 +40011.584,E4 +0.000} C_DIS
LIN {X -183.899,Y +1134.873,Z +0.000,A -10.372,E1 -42.805,E3 +40021.590,E4 +0.000} C_DIS
LIN {X -179.711,Y +1140.065,Z +0.000,A -15.940,E1 -40.393,E3 +40032.376,E4 +0.000} C_DIS
LIN {X -176.763,Y +1143.197,Z +0.000,A -18.748,E1 -38.674,E3 +40040.114,E4 +0.000} C_DIS
LIN {X -172.185,Y +1147.423,Z +0.000,A -19.971,E1 -36.175,E3 +40052.844,E4 +0.000} C_DIS
LIN {X -165.999,Y +1152.127,Z +0.000,A -20.000,E1 -32.027,E3 +40072.602,E4 +0.000} C_DIS
LIN {X -160.138,Y +1155.667,Z +0.000,A -20.000,E1 -26.368,E3 +40096.972,E4 +0.000} C_DIS
LIN {X -155.625,Y +1157.756,Z +0.000,A -20.000,E1 -19.505,E3 +40125.648,E4 +0.000} C_DIS
LIN {X -153.552,Y +1158.113,Z +0.000,A -20.000,E1 -11.113,E3 +40161.399,E4 +0.000} C_DIS
LIN {X -156.311,Y +1155.540,Z +0.000,A -20.000,E1 -0.839,E3 +40204.759,E4 +0.000} C_DIS
LIN {X -161.281,Y +1151.851,Z +0.000,A -20.000,E1 +7.737,E3 +40234.658,E4 +0.000} C_DIS
LIN {X -167.493,Y +1147.157,Z +0.000,A -20.000,E1 +16.195,E3 +40259.097,E4 +0.000} C_DIS
LIN {X -173.235,Y +1142.221,Z +0.000,A -20.000,E1 +22.930,E3 +40276.399,E4 +0.000} C_DIS
LIN {X -181.123,Y +1133.734,Z +0.000,A -20.000,E1 +30.868,E3 +40297.155,E4 +0.000} C_DIS
LIN {X -189.654,Y +1120.856,Z +0.000,A -20.000,E1 +39.018,E3 +40319.169,E4 +0.000} C_DIS
LIN {X -195.246,Y +1107.046,Z +0.000,A -20.000,E1 +44.515,E3 +40337.071,E4 +0.000} C_DIS
LIN {X -198.051,Y +1092.368,Z +0.000,A -20.000,E1 +47.947,E3 +40353.597,E4 +0.000} C_DIS
LIN {X -198.143,Y +1081.370,Z +0.000,A -19.806,E1 +49.153,E3 +40365.458,E4 +0.000} C_DIS
LIN {X -197.177,Y +1073.569,Z +0.000,A -17.356,E1 +49.162,E3 +40374.042,E4 +0.000} C_DIS
LIN {X -195.448,Y +1066.139,Z +0.000,A -12.154,E1 +48.512,E3 +40382.637,E4 +0.000} C_DIS
LIN {X -193.346,Y +1058.941,Z +0.000,A -7.133,E1 +47.724,E3 +40391.517,E4 +0.000} C_DIS
LIN {X -191.781,Y +1050.839,Z +0.000,A -3.715,E1 +47.274,E3 +40401.850,E4 +0.000} C_DIS
LIN {X -190.795,Y +1039.355,Z +0.000,A -0.983,E1 +46.842,E3 +40416.510,E4 +0.000} C_DIS
LIN {X -190.395,Y +1028.856,Z +0.000,A -0.089,E1 +46.598,E3 +40429.904,E4 +0.000} C_DIS
LIN {X -190.239,Y +1018.851,Z +0.000,A -0.004,E1 +46.529,E3 +40442.672,E4 +0.000} C_DIS
LIN {X -190.161,Y +1004.975,Z +0.000,A +0.000,E1 +46.506,E3 +40460.386,E4 +0.000} C_DIS
LIN {X -190.142,Y +412.853,Z +0.000,A +0.000,E1 +46.501,E3 +41216.592,E4 +0.000} C_DIS
LIN {X -190.147,Y +401.077,Z +0.000,A +0.000,E1 +46.499,E3 +41231.633,E4 +0.000} C_DIS
LIN {X -190.159,Y +390.929,Z +0.000,A +0.000,E1 +46.494,E3 +41244.599,E4 +0.000} C_DIS
LIN {X -190.174,Y +383.973,Z +0.000,A +0.000,E1 +46.484,E3 +41253.492,E4 +0.000} C_DIS
LIN {X -190.200,Y +373.815,Z +0.000,A +0.000,E1 +46.448,E3 +41266.497,E4 +0.000} C_DIS
LIN {X -190.154,Y +361.003,Z +0.000,A +0.000,E1 +46.303,E3 +41282.991,E4 +0.000} C_DIS
LIN {X -189.772,Y +350.660,Z +0.000,A +0.049,E1 +45.996,E3 +41296.530,E4 +0.000} C_DIS
LIN {X -189.325,Y +346.917,Z +0.000,A +0.243,E1 +45.771,E3 +41301.599,E4 +0.000} C_DIS
LIN {X -188.196,Y +342.754,Z +0.000,A +1.966,E1 +45.249,E3 +41307.607,E4 +0.000} C_DIS
LIN {X -185.199,Y +337.023,Z +0.000,A +6.630,E1 +43.793,E3 +41316.981,E4 +0.000} C_DIS
LIN {X -181.141,Y +331.596,Z +0.000,A +12.274,E1 +41.569,E3 +41327.541,E4 +0.000} C_DIS
LIN {X -176.762,Y +326.804,Z +0.000,A +17.560,E1 +38.898,E3 +41338.965,E4 +0.000} C_DIS
LIN {X -172.184,Y +322.578,Z +0.000,A +19.859,E1 +36.197,E3 +41351.695,E4 +0.000} C_DIS
LIN {X -165.998,Y +317.874,Z +0.000,A +20.000,E1 +32.027,E3 +41371.453,E4 +0.000} C_DIS
LIN {X -160.137,Y +314.334,Z +0.000,A +20.000,E1 +26.368,E3 +41395.822,E4 +0.000} C_DIS
LIN {X -155.624,Y +312.245,Z +0.000,A +20.000,E1 +19.506,E3 +41424.498,E4 +0.000} C_DIS
LIN {X -153.557,Y +311.879,Z +0.000,A +20.000,E1 +11.113,E3 +41460.253,E4 +0.000} C_DIS
LIN {X -155.320,Y +313.348,Z +0.000,A +20.000,E1 +3.401,E3 +41493.437,E4 +0.000} C_DIS
LIN {X -160.005,Y +315.804,Z +0.000,A +20.000,E1 -4.720,E3 +41523.815,E4 +0.000} C_DIS
LIN {X -164.504,Y +318.255,Z +0.000,A +20.000,E1 -10.663,E3 +41543.184,E4 +0.000} C_DIS
LIN {X -170.340,Y +322.684,Z +0.000,A +20.000,E1 -17.457,E3 +41563.216,E4 +0.000} C_DIS
LIN {X -175.568,Y +329.106,Z +0.000,A +20.000,E1 -24.747,E3 +41580.450,E4 +0.000} C_DIS
LIN {X -184.074,Y +340.065,Z +0.000,A +20.000,E1 -33.664,E3 +41603.390,E4 +0.000} C_DIS
LIN {X -190.779,Y +351.388,Z +0.000,A +20.000,E1 -40.083,E3 +41621.168,E4 +0.000} C_DIS
LIN {X -195.254,Y +362.955,Z +0.000,A +20.000,E1 -44.515,E3 +41635.921,E4 +0.000} C_DIS
LIN {X -197.754,Y +374.780,Z +0.000,A +20.000,E1 -47.450,E3 +41649.343,E4 +0.000} C_DIS
LIN {X -198.310,Y +383.215,Z +0.000,A +19.956,E1 -48.698,E3 +41658.467,E4 +0.000} C_DIS
LIN {X -197.912,Y +391.275,Z +0.000,A +18.601,E1 -49.158,E3 +41667.185,E4 +0.000} C_DIS
LIN {X -196.679,Y +398.944,Z +0.000,A +13.989,E1 -48.784,E3 +41675.739,E4 +0.000} C_DIS
LIN {X -194.742,Y +406.288,Z +0.000,A +8.476,E1 -48.001,E3 +41684.422,E4 +0.000} C_DIS
LIN {X -192.748,Y +413.472,Z +0.000,A +3.905,E1 -47.267,E3 +41693.432,E4 +0.000} C_DIS
LIN {X -191.781,Y +419.162,Z +0.000,A +1.739,E1 -46.975,E3 +41700.700,E4 +0.000} C_DIS
